	// ************* HMI - Show machine status on main screen ************* //
	IF ("dbUnit".Unit[1].Regime=0) AND NOT "dbUnit".Unit[1].StartStop THEN 
	  "dbUnit".Unit[1].Status     := 1;
	ELSIF ("dbUnit".Unit[1].Regime=0) AND "dbUnit".Unit[1].StartStop THEN 
	  "dbUnit".Unit[1].Status     := 2;
	ELSIF ("dbUnit".Unit[1].Regime>=1) AND NOT "dbUnit".Unit[1].StartStop THEN 
	  "dbUnit".Unit[1].Status     := 3;
	ELSIF ("dbUnit".Unit[1].Regime>=1) AND "dbUnit".Unit[1].StartStop THEN 
	  "dbUnit".Unit[1].Status     := 4;
	ELSIF ("dbUnit".Unit[1].Regime=0) AND ((NOT "ph_Helix_1_DB".InitPosition AND ("ph_Helix_1_DB".CurrentStep > 1 AND "ph_Helix_1_DB".CurrentStep <=2)) OR
	(NOT "ph_LegsShifter_2_DB".InitPosition AND ("ph_LegsShifter_2_DB".CurrentStep > 2 AND "ph_LegsShifter_2_DB".CurrentStep <=3))) THEN
	  "dbUnit".Unit[1].Status     := 5;
	END_IF;
	(*
	1-IZBRAN AVTOMATSKI NAČIN DELOVANJA
	2-AVTOMATSKI NAČIN AKTIVIRAN
	3-IZBRAN ROČNI NAČIN DELOVANJA
	4-ROČNI NAČIN AKTIVIRAN
	5-NAPRAVA NI V IZHODIŠČU
	*)
	// ************* HMI - Show machine status on main screen ************* //
	
	// ************* HMI - Animate HMI button ************* //
	IF "op_ButtonHelix_3_DB".AlarmPresent OR "ph_Helix_1_DB".AlarmPresent OR "ph_LegsShifter_2_DB".AlarmPresent THEN
	  "dbUnit".Unit[1].AlarmsPresent := True;
	ELSE
	  "dbUnit".Unit[1].AlarmsPresent := False;
	END_IF;
	// ************* HMI - Animate HMI button  ************* //
	
	// ************* HMI - BEGIN - Select screen  ************* //
	IF "dbUnit".Unit[1].Regime = 1 AND "dbUnit".Unit[1].StartStop THEN
	  (* NOT IN FUNCTION
	  IF "dbHMIUser".HMICurrScreen = 1 THEN
	    "dbHMIUser".SetTargetHMIScreen    := 2;
	  END_IF;
	  *)
	  IF ("dbHMIUser".HMICurrScreen <> 1) THEN 
	    ; // "dbHMIUser".SetTargetHMIScreen  := 0;
	  END_IF;
	END_IF;
	IF (NOT "dbUnit".Unit[1].StartStop) THEN
	  "dbHMIUser".SetTargetHMIScreen  := 0;
	END_IF;
	"dbHMIUser".HMICurrScreen_OLD := "dbHMIUser".HMICurrScreen;
	// ************* HMI - END - Select screen  ************* //
	
	// ************* HMI - BEGIN - Fill system param  ************* //
	"dbDigitalSensors".KONCNA_POZICIJA_VIJACENJA_DES_NAZAJ.FilterTime       := "dbSystemParam".KONCNA_POZICIJA_VIJACENJA_DES_NAZAJ_FilterTime;
	"dbDigitalSensors".KONCNA_POZICIJA_VIJACENJA_DES_NAPREJ.FilterTime      := "dbSystemParam".KONCNA_POZICIJA_VIJACENJA_DES_NAPREJ_FilterTime;
	"dbDigitalSensors".KONCNA_POZICIJA_VIJACENJA_LEVO_NAZAJ.FilterTime      := "dbSystemParam".KONCNA_POZICIJA_VIJACENJA_LEVO_NAZAJ_FilterTime;
	"dbDigitalSensors".KONCNA_POZICIJA_VIJACENJA_LEVO_NAPREJ.FilterTime     := "dbSystemParam".KONCNA_POZICIJA_VIJACENJA_DES_NAPREJ_FilterTime;
	"op_ButtonHelix_3_DB".DlyTimeToStart_TRAK_VIJAC := "dbSystemParam".DlyTimeToStart_TRAK_VIJAC*10;
	"op_ButtonHelix_3_DB".DlyTimeToStop_TRAK_VIJAC  := "dbSystemParam".DlyTimeToStop_TRAK_VIJAC*10;
	"op_ButtonHelix_3_DB".DlyTimeToStart_VIBRO      := "dbSystemParam".DlyTimeToStart_VIBRO*10;
	"op_ButtonHelix_3_DB".DlyTimeToStop_VIBRO       := "dbSystemParam".DlyTimeToStop_VIBRO*10;
	"dbTimers".Num[8].PRE                           := "dbSystemParam".StandbyTimeTrakaVijac*10*60; // On HMI in unit [min],
	"op_ButtonHelix_3_DB".DlyTimeForAlarmAddNewHelix := "dbSystemParam".DlyTimeForAlarmAddNewHelix * 10;
	// ************* HMI - END - Fill system param  ************* //
	
	// ************* BEGIN - Stop running trak vijačnika, if helix is no more in execution  ************* //
	// See above line "dbTimers".Num[8].PRE                           := "dbSystemParam".StandbyTimeTrakaVijac*10*60; // On HMI in unit [min]
	"dbTimers".Num[8].EE := "dbMotors".VKLOP_M_TRAKA_VIJACNIKA.XS;
	"dbTimers".Num[8].RS := "ph_Helix_1_DB".MovingUPDOWN_Activated;
	
	IF "dbTimers".Num[8].EE AND "dbTimers".Num[8].DN THEN
	  "dbTimers".Num[8].EE := False;
	  "dbTimers".Num[8].DN := False;
	  "dbTimers".Num[8].RS := False;
	  
	  "dbUnit".Unit[1].StartStop := False;
	END_IF;
	// ************* END - Stop running trak vijačnika, if helix is no more in execution  ************* //
END_FUNCTION

FUNCTION "fcDigitalValves" : Void
{ S7_Optimized_Access := 'FALSE' }
VERSION : 0.1
   VAR_TEMP 
      DigitalValveTime : Byte;
   END_VAR


BEGIN
	// Short summary:
	(*
	  Digital valves filter time set, output write and function call
	*)
	// 
	//**********************************************************************
	// Revision control:
	//----------------------------------------------------------------------
	// Use only for revisions of original code
	// V0.01
	// Description of revision
	
	//----------------------------------------------------------------------
	// Comments:
	(*
	  Every change in the code is documented with following:
	  // CCC-yyymmdd: .....
	  yyyy year when change was made
	  mm   month when change was made
	  dd   day when change was made
	  CCC  authors initials
	*)
	
	(*
	- VPENJANJE: V18
	- CENTRIRANJE: V7, V10, V14, V17
	- STOP VIJACENJA ZADAJ: V5, V12
	- LOCEVANJE VIJACENJA: V4, V11
	- LOCEVANJE DRCA: V2, V3
	- DVIG/SPUST VIJACENJA: V6, V9, V13, V16
	*)
	
	//**********************************************************************
	#DigitalValveTime := 10; // Filter time =0. For digital valve is used throught digital sensor with filter time for ."InputF"
	//----------------------------------------------------------------------
	//  set initial values
	"dbDigitalValves".Y17_RotCilipozDesno.FilterTime    := 15;
	"dbDigitalValves".Y18_RotCilipozLevo.FilterTime     := 15;
	"dbDigitalValves".Y2_VijaDesZad_Dvig.FilterTime     := 50;
	"dbDigitalValves".Y3_VijaDesSpr_Dvig.FilterTime     := 50;
	"dbDigitalValves".Y4_VijaLevZad_Dvig.FilterTime     := 50;
	"dbDigitalValves".Y5_VijaLevSpr_Dvig.FilterTime     := 50;
	"dbDigitalValves".Y6_DrcaLocev_Des.FilterTime       := #DigitalValveTime;
	"dbDigitalValves".Y7_DrcaLocev_Lev.FilterTime       := #DigitalValveTime;
	"dbDigitalValves".Y8_VijaLocev_Des.FilterTime       := #DigitalValveTime;
	"dbDigitalValves".Y9_VijaStop_DesZad.FilterTime     := #DigitalValveTime;
	"dbDigitalValves".Y10_Centri_DesZad.FilterTime      := #DigitalValveTime;
	"dbDigitalValves".Y11_Centri_DesSpr.FilterTime      := #DigitalValveTime;
	"dbDigitalValves".Y12_VijaLocev_Lev.FilterTime      := #DigitalValveTime;
	"dbDigitalValves".Y13_VijaStop_LevZad.FilterTime    := #DigitalValveTime;
	"dbDigitalValves".Y14_Centri_LevZad.FilterTime      := #DigitalValveTime;
	"dbDigitalValves".Y15_Centri_LevSpr.FilterTime      := #DigitalValveTime;
	"dbDigitalValves".Y16_VpenjanjeDna.FilterTime       := 30;
	"dbDigitalValves".SEMAFOR_ZELENA.FilterTime         := #DigitalValveTime;
	"dbDigitalValves".SEMAFOR_RUMENA.FilterTime         := #DigitalValveTime;
	"dbDigitalValves".SEMAFOR_RDECA.FilterTime          := #DigitalValveTime;
	
	"dbDigitalValves".Y17_RotCilipozDesno.Invert       := False;
	"dbDigitalValves".Y18_RotCilipozLevo.Invert        := False;
	"dbDigitalValves".Y2_VijaDesZad_Dvig.Invert       := False;
	"dbDigitalValves".Y3_VijaDesSpr_Dvig.Invert       := False;
	"dbDigitalValves".Y4_VijaLevZad_Dvig.Invert      := False;
	"dbDigitalValves".Y5_VijaLevSpr_Dvig.Invert      := False;
	"dbDigitalValves".Y6_DrcaLocev_Des.Invert         := False;
	"dbDigitalValves".Y7_DrcaLocev_Lev.Invert         := False;
	"dbDigitalValves".Y8_VijaLocev_Des.Invert         := False;
	"dbDigitalValves".Y9_VijaStop_DesZad.Invert       := False;
	"dbDigitalValves".Y10_Centri_DesZad.Invert         := False;
	"dbDigitalValves".Y11_Centri_DesSpr.Invert        := False;
	"dbDigitalValves".Y12_VijaLocev_Lev.Invert        := False;
	"dbDigitalValves".Y13_VijaStop_LevZad.Invert      := False;
	"dbDigitalValves".Y14_Centri_LevZad.Invert        := False;
	"dbDigitalValves".Y15_Centri_LevSpr.Invert        := False;
	"dbDigitalValves".Y16_VpenjanjeDna.Invert         := False;
	"dbDigitalValves".SEMAFOR_ZELENA.Invert           := False;
	"dbDigitalValves".SEMAFOR_RUMENA.Invert           := False;
	"dbDigitalValves".SEMAFOR_RDECA.Invert            := False;
	
	"dbDigitalValves".Y17_RotCilipozDesno.AlarmAck       := "AlarmAck";
	"dbDigitalValves".Y18_RotCilipozLevo.AlarmAck        := "AlarmAck";
	"dbDigitalValves".Y2_VijaDesZad_Dvig.AlarmAck       := "AlarmAck";
	"dbDigitalValves".Y3_VijaDesSpr_Dvig.AlarmAck       := "AlarmAck";
	"dbDigitalValves".Y4_VijaLevZad_Dvig.AlarmAck      := "AlarmAck";
	"dbDigitalValves".Y5_VijaLevSpr_Dvig.AlarmAck      := "AlarmAck";
	"dbDigitalValves".Y6_DrcaLocev_Des.AlarmAck         := "AlarmAck";
	"dbDigitalValves".Y7_DrcaLocev_Lev.AlarmAck         := "AlarmAck";
	"dbDigitalValves".Y8_VijaLocev_Des.AlarmAck         := "AlarmAck";
	"dbDigitalValves".Y9_VijaStop_DesZad.AlarmAck       := "AlarmAck";
	"dbDigitalValves".Y10_Centri_DesZad.AlarmAck         := "AlarmAck";
	"dbDigitalValves".Y11_Centri_DesSpr.AlarmAck        := "AlarmAck";
	"dbDigitalValves".Y12_VijaLocev_Lev.AlarmAck        := "AlarmAck";
	"dbDigitalValves".Y13_VijaStop_LevZad.AlarmAck      := "AlarmAck";
	"dbDigitalValves".Y14_Centri_LevZad.AlarmAck        := "AlarmAck";
	"dbDigitalValves".Y15_Centri_LevSpr.AlarmAck        := "AlarmAck";
	"dbDigitalValves".Y16_VpenjanjeDna.AlarmAck         := "AlarmAck";
	"dbDigitalValves".SEMAFOR_ZELENA.AlarmAck           := "AlarmAck";
	"dbDigitalValves".SEMAFOR_RUMENA.AlarmAck           := "AlarmAck";
	"dbDigitalValves".SEMAFOR_RDECA.AlarmAck            := "AlarmAck";
	
	// read GSL
	"dbDigitalValves".Y17_RotCilipozDesno.GSLEnable    := TRUE;
	"dbDigitalValves".Y17_RotCilipozDesno.GSL          := "dbDigitalSensors".ROTACIJSKI_CIL_SREDINA.InputF OR "dbDigitalValves".Y18_RotCilipozLevo.XS;
	"dbDigitalValves".Y18_RotCilipozLevo.GSLEnable     := TRUE;
	"dbDigitalValves".Y18_RotCilipozLevo.GSL           := "dbDigitalSensors".ROTACIJSKI_CIL_SREDINA.InputF OR "dbDigitalValves".Y17_RotCilipozDesno.XS;
	"dbDigitalValves".Y2_VijaDesZad_Dvig.GSLEnable    := True;
	"dbDigitalValves".Y2_VijaDesZad_Dvig.GSL          := "dbDigitalSensors".MESTO_VIJACENJE_DESNO_ZAD_DVIG_DOL.InputF;
	"dbDigitalValves".Y3_VijaDesSpr_Dvig.GSLEnable    := True;
	"dbDigitalValves".Y3_VijaDesSpr_Dvig.GSL          := "dbDigitalSensors".MESTO_VIJACENJE_DESNO_SPRED_DVIG_DOL.InputF;
	"dbDigitalValves".Y4_VijaLevZad_Dvig.GSLEnable   := True;
	"dbDigitalValves".Y4_VijaLevZad_Dvig.GSL         := "dbDigitalSensors".MESTO_VIJACENJE_LEVO_ZAD_DVIG_DOL.InputF;
	"dbDigitalValves".Y5_VijaLevSpr_Dvig.GSLEnable   := True;
	"dbDigitalValves".Y5_VijaLevSpr_Dvig.GSL         := "dbDigitalSensors".MESTO_VIJACENJE_LEVO_SPRED_DVIG_DOL.InputF;
	"dbDigitalValves".Y6_DrcaLocev_Des.GSLEnable      := True;
	"dbDigitalValves".Y6_DrcaLocev_Des.GSL            := "dbDigitalSensors".LOC_DRCA_DESNO_NAPREJ.InputF;
	"dbDigitalValves".Y7_DrcaLocev_Lev.GSLEnable      := True;
	"dbDigitalValves".Y7_DrcaLocev_Lev.GSL            := "dbDigitalSensors".LOC_DRCA_LEVO_NAPREJ.InputF;
	"dbDigitalValves".Y8_VijaLocev_Des.GSLEnable      := True;
	"dbDigitalValves".Y8_VijaLocev_Des.GSL            := "dbDigitalSensors".VIJACENJE_DESNO_1_NAPREJ.InputF;
	"dbDigitalValves".Y9_VijaStop_DesZad.GSLEnable    := True;
	"dbDigitalValves".Y9_VijaStop_DesZad.GSL          := "dbDigitalSensors".MESTO_VIJAC_STOP_DESNO_ZAD_NAPREJ.InputF;
	"dbDigitalValves".Y10_Centri_DesZad.GSLEnable      := True;
	"dbDigitalValves".Y10_Centri_DesZad.GSL            := "dbDigitalSensors".MESTO_VIJACENJE_DESNO_ZAD_CENT_NARAZEN.InputF;
	"dbDigitalValves".Y11_Centri_DesSpr.GSLEnable     := True;
	"dbDigitalValves".Y11_Centri_DesSpr.GSL           := "dbDigitalSensors".MESTO_VIJACENJE_DESNO_SPRED_CENT_NARAZEN.InputF;
	"dbDigitalValves".Y12_VijaLocev_Lev.GSLEnable     := True;
	"dbDigitalValves".Y12_VijaLocev_Lev.GSL           := "dbDigitalSensors".VIJACENJE_LEVO_1_NAPREJ.InputF;
	"dbDigitalValves".Y13_VijaStop_LevZad.GSLEnable   := True;
	"dbDigitalValves".Y13_VijaStop_LevZad.GSL         := "dbDigitalSensors".MESTO_VIJAC_STOP_LEVO_ZAD_NAPREJ.InputF;
	"dbDigitalValves".Y14_Centri_LevZad.GSLEnable     := True;
	"dbDigitalValves".Y14_Centri_LevZad.GSL           := "dbDigitalSensors".MESTO_VIJACENJE_LEVO_ZAD_CENT_NARAZEN.InputF;
	"dbDigitalValves".Y15_Centri_LevSpr.GSLEnable     := True;
	"dbDigitalValves".Y15_Centri_LevSpr.GSL           := "dbDigitalSensors".MESTO_VIJACENJE_LEVO_SPRED_CENT_NARAZEN.InputF;
	"dbDigitalValves".Y16_VpenjanjeDna.GSLEnable      := True;
	"dbDigitalValves".Y16_VpenjanjeDna.GSL            := "dbDigitalSensors".VPENJANJE_DNA_LEVO_ZADAJ_GOR.InputF AND "dbDigitalSensors".VPENJANJE_DNA_LEVO_SPREDAJ_GOR.InputF AND
	                                                     "dbDigitalSensors".VPENJANJE_DNA_DESNO_ZADAJ_GOR.InputF AND "dbDigitalSensors".VPENJANJE_DNA_DESNO_SPREDAJ_GOR.InputF;
	
	// read GSH
	"dbDigitalValves".Y17_RotCilipozDesno.GSHEnable    := TRUE;
	"dbDigitalValves".Y17_RotCilipozDesno.GSH          := "dbDigitalSensors".ROTACIJSKI_CIL_DESNO.InputF;
	"dbDigitalValves".Y18_RotCilipozLevo.GSHEnable     := True;
	"dbDigitalValves".Y18_RotCilipozLevo.GSH           := "dbDigitalSensors".ROTACIJSKI_CIL_LEVO.InputF;
	"dbDigitalValves".Y2_VijaDesZad_Dvig.GSHEnable    := FALSE;
	"dbDigitalValves".Y2_VijaDesZad_Dvig.GSH          := FALSE;
	"dbDigitalValves".Y3_VijaDesSpr_Dvig.GSHEnable    := FALSE;
	"dbDigitalValves".Y3_VijaDesSpr_Dvig.GSH          := FALSE;
	"dbDigitalValves".Y4_VijaLevZad_Dvig.GSHEnable   := FALSE;
	"dbDigitalValves".Y4_VijaLevZad_Dvig.GSH         := FALSE;
	"dbDigitalValves".Y5_VijaLevSpr_Dvig.GSHEnable   := False;
	"dbDigitalValves".Y5_VijaLevSpr_Dvig.GSH         := False;
	"dbDigitalValves".Y6_DrcaLocev_Des.GSHEnable      := True;
	"dbDigitalValves".Y6_DrcaLocev_Des.GSH            := "dbDigitalSensors".LOC_DRCA_DESNO_NAZAJ.InputF;
	"dbDigitalValves".Y7_DrcaLocev_Lev.GSHEnable      := True;
	"dbDigitalValves".Y7_DrcaLocev_Lev.GSH            := "dbDigitalSensors".LOC_DRCA_LEVO_NAZAJ.InputF;
	"dbDigitalValves".Y8_VijaLocev_Des.GSHEnable      := True;
	"dbDigitalValves".Y8_VijaLocev_Des.GSH            := "dbDigitalSensors".VIJACENJE_DESNO_1_NAZAJ.InputF;
	"dbDigitalValves".Y9_VijaStop_DesZad.GSHEnable    := True;
	"dbDigitalValves".Y9_VijaStop_DesZad.GSH          := "dbDigitalSensors".MESTO_VIJAC_STOP_DESNO_ZAD_NAZAJ.InputF;
	"dbDigitalValves".Y10_Centri_DesZad.GSHEnable      := True;
	"dbDigitalValves".Y10_Centri_DesZad.GSH            := "dbDigitalSensors".MESTO_VIJACENJE_DESNO_ZAD_CENT_SKUPAJ.InputF;
	"dbDigitalValves".Y11_Centri_DesSpr.GSHEnable     := True;
	"dbDigitalValves".Y11_Centri_DesSpr.GSH           := "dbDigitalSensors".MESTO_VIJACENJE_DESNO_SPRED_CENT_SKUPAJ.InputF;
	"dbDigitalValves".Y12_VijaLocev_Lev.GSHEnable     := True;
	"dbDigitalValves".Y12_VijaLocev_Lev.GSH           := "dbDigitalSensors".VIJACENJE_LEVO_1_NAZAJ.InputF;
	"dbDigitalValves".Y13_VijaStop_LevZad.GSHEnable   := True;
	"dbDigitalValves".Y13_VijaStop_LevZad.GSH         := "dbDigitalSensors".MESTO_VIJAC_STOP_LEVO_ZAD_NAZAJ.InputF;;
	"dbDigitalValves".Y14_Centri_LevZad.GSHEnable     := True;
	"dbDigitalValves".Y14_Centri_LevZad.GSH           := "dbDigitalSensors".MESTO_VIJACENJE_LEVO_ZAD_CENT_SKUPAJ.InputF;
	"dbDigitalValves".Y15_Centri_LevSpr.GSHEnable     := True;
	"dbDigitalValves".Y15_Centri_LevSpr.GSH           := "dbDigitalSensors".MESTO_VIJACENJE_LEVO_SPRED_CENT_SKUPAJ.InputF;
	"dbDigitalValves".Y16_VpenjanjeDna.GSHEnable      := True;
	"dbDigitalValves".Y16_VpenjanjeDna.GSH            := "dbDigitalSensors".VPENJANJE_DNA_LEVO_ZADAJ_DOL.InputF AND "dbDigitalSensors".VPENJANJE_DNA_LEVO_SPREDAJ_DOL.InputF AND
	                                                     "dbDigitalSensors".VPENJANJE_DNA_DESNO_ZADAJ_DOL.InputF AND "dbDigitalSensors".VPENJANJE_DNA_DESNO_SPREDAJ_DOL.InputF;
	
	// Reset Manual Regime, if selected AUTO regime on HMI
	//----------------------------------------------------------------------
	IF "dbUnit".Unit[1].Regime = 0 AND "dbUnit".Unit[1].StartStop THEN
	  "dbDigitalValves".Y17_RotCilipozDesno.ManON   := False;
	  "dbDigitalValves".Y18_RotCilipozLevo.ManON    := False;
	  "dbDigitalValves".Y2_VijaDesZad_Dvig.ManON    := False;
	  "dbDigitalValves".Y2_VijaDesZad_Dvig.ManON    := False;
	  "dbDigitalValves".Y3_VijaDesSpr_Dvig.ManON    := False;
	  "dbDigitalValves".Y3_VijaDesSpr_Dvig.ManON    := False;
	  "dbDigitalValves".Y4_VijaLevZad_Dvig.ManON    := False;
	  "dbDigitalValves".Y4_VijaLevZad_Dvig.ManON    := False;
	  "dbDigitalValves".Y5_VijaLevSpr_Dvig.ManON    := False;
	  "dbDigitalValves".Y5_VijaLevSpr_Dvig.ManON    := False;
	  "dbDigitalValves".Y6_DrcaLocev_Des.ManON      := False;
	  "dbDigitalValves".Y7_DrcaLocev_Lev.ManON      := False;
	  "dbDigitalValves".Y8_VijaLocev_Des.ManON      := False;
	  "dbDigitalValves".Y9_VijaStop_DesZad.ManON    := False;
	  "dbDigitalValves".Y10_Centri_DesZad.ManON     := False;
	  "dbDigitalValves".Y11_Centri_DesSpr.ManON     := False;
	  "dbDigitalValves".Y12_VijaLocev_Lev.ManON     := False;
	  "dbDigitalValves".Y13_VijaStop_LevZad.ManON   := False;
	  "dbDigitalValves".Y14_Centri_LevZad.ManON     := False;
	  "dbDigitalValves".Y15_Centri_LevSpr.ManON     := False;
	ELSIF "dbUnit".Unit[1].Regime = 1 AND NOT "dbUnit".Unit[1].StartStop THEN
	  "dbDigitalValves".Y17_RotCilipozDesno.ManON   := False;
	  "dbDigitalValves".Y18_RotCilipozLevo.ManON    := False;
	  "dbDigitalValves".Y2_VijaDesZad_Dvig.ManON    := False;
	  "dbDigitalValves".Y2_VijaDesZad_Dvig.ManON    := False;
	  "dbDigitalValves".Y3_VijaDesSpr_Dvig.ManON    := False;
	  "dbDigitalValves".Y3_VijaDesSpr_Dvig.ManON    := False;
	  "dbDigitalValves".Y4_VijaLevZad_Dvig.ManON    := False;
	  "dbDigitalValves".Y4_VijaLevZad_Dvig.ManON    := False;
	  "dbDigitalValves".Y5_VijaLevSpr_Dvig.ManON    := False;
	  "dbDigitalValves".Y5_VijaLevSpr_Dvig.ManON    := False;
	  "dbDigitalValves".Y6_DrcaLocev_Des.ManON      := False;
	  "dbDigitalValves".Y7_DrcaLocev_Lev.ManON      := False;
	  "dbDigitalValves".Y8_VijaLocev_Des.ManON      := False;
	  "dbDigitalValves".Y9_VijaStop_DesZad.ManON    := False;
	  "dbDigitalValves".Y10_Centri_DesZad.ManON     := False;
	  "dbDigitalValves".Y11_Centri_DesSpr.ManON     := False;
	  "dbDigitalValves".Y12_VijaLocev_Lev.ManON     := False;
	  "dbDigitalValves".Y13_VijaStop_LevZad.ManON   := False;
	  "dbDigitalValves".Y14_Centri_LevZad.ManON     := False;
	  "dbDigitalValves".Y15_Centri_LevSpr.ManON     := False;
	END_IF; 
	
	//----------------------------------------------------------------------
	// fc call
	"cmDigitalValve"(Regime := "dbUnit".Unit[1].Regime, Valve := "dbDigitalValves".Y17_RotCilipozDesno);
	"cmDigitalValve"(Regime := "dbUnit".Unit[1].Regime, Valve := "dbDigitalValves".Y18_RotCilipozLevo);
	"cmDigitalValve"(Regime := "dbUnit".Unit[1].Regime, Valve := "dbDigitalValves".Y2_VijaDesZad_Dvig);
	"cmDigitalValve"(Regime := "dbUnit".Unit[1].Regime, Valve := "dbDigitalValves".Y3_VijaDesSpr_Dvig);
	"cmDigitalValve"(Regime := "dbUnit".Unit[1].Regime, Valve := "dbDigitalValves".Y4_VijaLevZad_Dvig);
	"cmDigitalValve"(Regime := "dbUnit".Unit[1].Regime, Valve := "dbDigitalValves".Y5_VijaLevSpr_Dvig);
	"cmDigitalValve"(Regime := "dbUnit".Unit[1].Regime, Valve := "dbDigitalValves".Y6_DrcaLocev_Des);
	"cmDigitalValve"(Regime := "dbUnit".Unit[1].Regime, Valve := "dbDigitalValves".Y7_DrcaLocev_Lev);
	"cmDigitalValve"(Regime := "dbUnit".Unit[1].Regime, Valve := "dbDigitalValves".Y8_VijaLocev_Des);
	"cmDigitalValve"(Regime := "dbUnit".Unit[1].Regime, Valve := "dbDigitalValves".Y9_VijaStop_DesZad);
	"cmDigitalValve"(Regime := "dbUnit".Unit[1].Regime, Valve := "dbDigitalValves".Y10_Centri_DesZad);
	"cmDigitalValve"(Regime := "dbUnit".Unit[1].Regime, Valve := "dbDigitalValves".Y11_Centri_DesSpr);
	"cmDigitalValve"(Regime := "dbUnit".Unit[1].Regime, Valve := "dbDigitalValves".Y12_VijaLocev_Lev);
	"cmDigitalValve"(Regime := "dbUnit".Unit[1].Regime, Valve := "dbDigitalValves".Y13_VijaStop_LevZad);
	"cmDigitalValve"(Regime := "dbUnit".Unit[1].Regime, Valve := "dbDigitalValves".Y14_Centri_LevZad);
	"cmDigitalValve"(Regime := "dbUnit".Unit[1].Regime, Valve := "dbDigitalValves".Y15_Centri_LevSpr);
	"cmDigitalValve"(Regime := "dbUnit".Unit[1].Regime, Valve := "dbDigitalValves".Y16_VpenjanjeDna);
	"cmDigitalValve"(Regime := "dbUnit".Unit[1].Regime, Valve := "dbDigitalValves".SEMAFOR_ZELENA);
	"cmDigitalValve"(Regime := "dbUnit".Unit[1].Regime, Valve := "dbDigitalValves".SEMAFOR_RUMENA);
	"cmDigitalValve"(Regime := "dbUnit".Unit[1].Regime, Valve := "dbDigitalValves".SEMAFOR_RDECA);
	
	//----------------------------------------------------------------------
	//  write output
	"dbPDO".Y17_RotCilipozDesno    := "dbDigitalValves".Y17_RotCilipozDesno.XS;
	"dbPDO".Y18_RotCilipozLevo     := "dbDigitalValves".Y18_RotCilipozLevo.XS;
	"dbPDO".Y2_VijaDesZad_Dvig    := "dbDigitalValves".Y2_VijaDesZad_Dvig.XS;
	"dbPDO".Y2_VijaDesZad_Spust   := NOT "dbDigitalValves".Y2_VijaDesZad_Dvig.XS;
	"dbPDO".Y3_VijaDesSpr_Dvig    := "dbDigitalValves".Y3_VijaDesSpr_Dvig.XS;
	"dbPDO".Y3_VijaDesSpr_Spust   := NOT "dbDigitalValves".Y3_VijaDesSpr_Dvig.XS;
	"dbPDO".Y4_VijaLevZad_Dvig   := "dbDigitalValves".Y4_VijaLevZad_Dvig.XS;
	"dbPDO".Y4_VijaLevZad_Spust  := NOT "dbDigitalValves".Y4_VijaLevZad_Dvig.XS;
	"dbPDO".Y5_VijaLevSpr_Dvig   := "dbDigitalValves".Y5_VijaLevSpr_Dvig.XS;
	"dbPDO".Y5_VijaLevSpr_Spust  := NOT "dbDigitalValves".Y5_VijaLevSpr_Dvig.XS;
	"dbPDO".Y6_DrcaLocev_Des      := "dbDigitalValves".Y6_DrcaLocev_Des.XS;
	"dbPDO".Y7_DrcaLocev_Lev      := "dbDigitalValves".Y7_DrcaLocev_Lev.XS;
	"dbPDO".Y8_VijaLocev_Des      := "dbDigitalValves".Y8_VijaLocev_Des.XS;
	"dbPDO".Y9_VijaStop_DesZad    := "dbDigitalValves".Y9_VijaStop_DesZad.XS;
	"dbPDO".Y10_Centri_DesZad      := "dbDigitalValves".Y10_Centri_DesZad.XS;
	"dbPDO".Y11_Centri_DesSpr     := "dbDigitalValves".Y11_Centri_DesSpr.XS;
	"dbPDO".Y12_VijaLocev_Lev     := "dbDigitalValves".Y12_VijaLocev_Lev.XS;
	"dbPDO".Y13_VijaStop_LevZad   := "dbDigitalValves".Y13_VijaStop_LevZad.XS;
	"dbPDO".Y14_Centri_LevZad     := "dbDigitalValves".Y14_Centri_LevZad.XS;
	"dbPDO".Y15_Centri_LevSpr     := "dbDigitalValves".Y15_Centri_LevSpr.XS;
	"dbPDO".Y16_VpenjanjeDna      := "dbDigitalValves".Y16_VpenjanjeDna.XS;
	
	"dbDO".SEMAFOR_ZELENA         := "dbDigitalValves".SEMAFOR_ZELENA.XS;
	"dbDO".SEMAFOR_RUMENA         := "dbDigitalValves".SEMAFOR_RUMENA.XS;
	"dbDO".SEMAFOR_RDECA          := "dbDigitalValves".SEMAFOR_RDECA.XS;
END_FUNCTION

FUNCTION "cmDigitalValve" : Void
{ S7_Optimized_Access := 'FALSE' }
VERSION : 0.1
   VAR_IN_OUT 
      Regime : USInt;
      Valve : "udtDigitalValve";
   END_VAR

   VAR_TEMP 
      tmpTimer : Int;
      tmpTimerDelay : Int;
   END_VAR

   VAR CONSTANT 
      AlarmAutoResetDly : UInt := 50;
   END_VAR


BEGIN
	// ALARMING
	#tmpTimer := CHAR_TO_INT(BYTE_TO_CHAR(#Valve.Timer1));
	#tmpTimerDelay := CHAR_TO_INT(BYTE_TO_CHAR(#Valve.FilterTime));
	
	IF (NOT #Valve.GSLEnable AND NOT #Valve.GSHEnable) THEN
	    #Valve.Alarm := FALSE;
	    #tmpTimer := 0;
	END_IF;
	
	IF ((#Valve.GSLEnable AND NOT #Valve.GSHEnable) AND ((NOT #Valve.SCADAVis AND NOT #Valve.GSL) OR (#Valve.SCADAVis AND #Valve.GSL))) OR
	    ((NOT #Valve.GSLEnable AND #Valve.GSHEnable) AND ((#Valve.SCADAVis AND NOT #Valve.GSH) OR (NOT #Valve.SCADAVis AND #Valve.GSH))) OR
	    ((#Valve.GSLEnable AND #Valve.GSHEnable) AND ((#Valve.SCADAVis AND (#Valve.GSL OR NOT #Valve.GSH)) OR (NOT #Valve.SCADAVis AND (NOT #Valve.GSL OR #Valve.GSH)))) THEN
	    
	    IF (NOT #Valve.Alarm) AND "100msOSR" AND (#tmpTimer <= #tmpTimerDelay) THEN
	        #tmpTimer := #tmpTimer + 1;
	        IF #tmpTimer >= #tmpTimerDelay THEN
	            #Valve.Alarm := TRUE;
	            #Valve.GSLAlarm := ((#Valve.GSLEnable) AND ((NOT #Valve.SCADAVis AND NOT #Valve.GSL) OR (#Valve.SCADAVis AND #Valve.GSL)));
	            #Valve.GSHAlarm := ((#Valve.GSHEnable) AND ((#Valve.SCADAVis AND NOT #Valve.GSH) OR (NOT #Valve.SCADAVis AND #Valve.GSH)));
	            #tmpTimer := 0;
	        END_IF;
	    END_IF;
	    IF (#Valve.Alarm) THEN
	        #tmpTimer := 0;
	    END_IF;
	// ELSIF ((#Valve.GSLEnable AND NOT #Valve.GSHEnable) AND (NOT #Valve.SCADAVis AND #Valve.GSL) OR // 20210429_PRA
	   ELSIF ((#Valve.GSLEnable AND NOT #Valve.GSHEnable) AND (NOT #Valve.SCADAVis AND #Valve.GSL) OR #Valve.SCADAVis) OR // 20210429_PRA-added to reset timer when valve activated
	    ((NOT #Valve.GSLEnable AND #Valve.GSHEnable) AND (#Valve.SCADAVis AND #Valve.GSH)) OR
	    ((#Valve.GSLEnable AND #Valve.GSHEnable) AND ((#Valve.SCADAVis AND #Valve.GSH) OR (NOT #Valve.SCADAVis AND #Valve.GSL))) THEN
	   
	    #tmpTimer := 0;
	    ;
	    (*
	    IF (#Valve.Alarm) AND "100msOSR" AND (#tmpTimer < AlarmAutoResetDly) THEN // Auto-reset of the alarm after 5 seconds
	        #tmpTimer := #tmpTimer + 1;
	        IF #tmpTimer >= AlarmAutoResetDly THEN
	            #Valve.Alarm := FALSE;
	            #Valve.GSLAlarm := FALSE;
	            #Valve.GSHAlarm := FALSE;
	            #tmpTimer := 0;
	        END_IF;
	    END_IF;
	    IF (NOT #Valve.Alarm) THEN
	        #tmpTimer := 0;
	    END_IF;
	    *)
	END_IF;
	
	//  ALARMING MODULE
	IF #Valve.AlarmAck THEN
	    #Valve.Alarm := FALSE;
	    #Valve.GSLAlarm := FALSE;
	    #Valve.GSHAlarm := FALSE;
	    #Valve.AlarmAck := FALSE;
	    
	    #tmpTimer := 0;
	END_IF;
	
	#Valve.Timer1 := CHAR_TO_BYTE(INT_TO_CHAR(#tmpTimer));
	
	//----------------------------------------------------------------------
	//  OUTPUT   
	#Valve.XS := FALSE;
	
	IF #Regime = 0 THEN
	    #Valve.ManON := FALSE;
	    #Valve.ManOFF := FALSE;
	    #Valve.XS := #Valve.AutoON;
	    #Valve.HMICmd := false;
	ELSIF #Regime > 0 THEN
	    IF #Valve.HMICmd THEN
	        IF NOT #Valve.SCADAVis THEN
	            #Valve.ManON := true;
	            #Valve.ManOFF := false;
	        END_IF;
	        IF #Valve.SCADAVis THEN
	            #Valve.ManON := false;
	            #Valve.ManOFF := true;
	        END_IF;
	        #Valve.HMICmd := false;
	    END_IF;
	    #Valve.XS := (#Valve.AutoON AND NOT #Valve.ManON AND NOT #Valve.ManOFF) OR (#Valve.ManON AND NOT #Valve.ManOFF);
	END_IF;
	
	//----------------------------------------------------------------------
	//  MANUAL BIT
	#Valve.Manual := #Valve.ManON OR #Valve.ManOFF;
	
	//----------------------------------------------------------------------
	//  INTERLOCK
	IF (#Valve.Interlock AND #Regime < 2) THEN
	    #Valve.XS := FALSE;
	END_IF;
	
	//----------------------------------------------------------------------
	//  NORMALY OPEN VALVES
	IF (#Valve.Invert) THEN
	    #Valve.XS := NOT (#Valve.XS);
	END_IF;
	
	//----------------------------------------------------------------------
	// SCADA VIS flag
	IF #Valve.Invert = TRUE THEN
	    #Valve.SCADAVis := NOT (#Valve.XS);
	ELSE
	    #Valve.SCADAVis := #Valve.XS;
	END_IF;
	
	//----------------------------------------------------------------------
	// Valve Status
	IF NOT #Valve.SCADAVis THEN
	    #Valve.Status := 0;
	END_IF;
	IF #Valve.SCADAVis THEN
	    #Valve.Status := 1;
	END_IF;
	IF #Valve.Alarm THEN
	    #Valve.Status := 2;
	END_IF;
	(*
	IF #Valve.GSLAlarm THEN
	    #Valve.Status := 3;
	END_IF;
	IF #Valve.GSHAlarm THEN
	    #Valve.Status := 4;
	END_IF;
	*)
	
	
END_FUNCTION

FUNCTION "fcMotors" : Void
{ S7_Optimized_Access := 'TRUE' }
VERSION : 0.1
   VAR CONSTANT 
      CONST_FILTER_TIME_EA : USInt := 10;
      CONST_FILTER_TIME_FSL : USInt := 50;
   END_VAR


BEGIN
	// Short summary:
	(*
	  fcMotors - call motors
	*)
	// 
	//**********************************************************************
	// Revision control:
	//----------------------------------------------------------------------
	// Use only for revisions of original code
	// V0.01
	// Description of revision
	
	//----------------------------------------------------------------------
	// Comments:
	(*
	  Every change in the code is documented with following:
	  // CCC-yyymmdd: .....
	  yyyy year when change was made
	  mm   month when change was made
	  dd   day when change was made
	  CCC  authors initials
	*)
	//**********************************************************************
	
	//  set motor parameters
	"dbMotors".VKLOP_M_TRACNEGA_TRANS_NOGIC.MaxEng  := 100.0; // Max motor RPM
	"dbMotors".VKLOP_M_TRACNEGA_TRANS_NOGIC.MinEng  := 0.0;   // Min motor RPM
	"dbMotors".VKLOP_M_TRACNEGA_TRANS_NOGIC.ESA     := NOT "dbDigitalSensors".BIMETAL_TRANSPORTA_NOGIC_IZKLJUCIL.InputF;
	"dbMotors".VKLOP_M_TRACNEGA_TRANS_NOGIC.EA      := "dbDO".VKLOP_M_TRACNEGA_TRANS_NOGIC;
	"dbMotors".VKLOP_M_TRACNEGA_TRANS_NOGIC.FSL     := "dbDO".VKLOP_M_TRACNEGA_TRANS_NOGIC;
	"dbMotors".VKLOP_M_TRACNEGA_TRANS_NOGIC.AlarmAck := "AlarmAck";
	// "dbDO". := "dbMotors".M_TRACNEGA_TRANSPORTA.ResetFCAlarm;
	"dbMotors".VKLOP_M_TRACNEGA_TRANS_NOGIC.FILTER_TIME_EA  := #CONST_FILTER_TIME_EA;   // 10 sec
	"dbMotors".VKLOP_M_TRACNEGA_TRANS_NOGIC.FILTER_TIME_FSL := #CONST_FILTER_TIME_FSL;  // 50 sec
	
	"dbMotors".M1_ZADAJ_DESNO.MaxEng  := 100.0; // Max motor RPM
	"dbMotors".M1_ZADAJ_DESNO.MinEng  := 0.0;   // Min motor RPM
	"dbMotors".M1_ZADAJ_DESNO.ESA     := "dbDigitalSensors".FR_MOTORJA1_ZADAJ_DESNO_READY.InputF;
	"dbMotors".M1_ZADAJ_DESNO.EA      := "dbMotors".M1_ZADAJ_DESNO.XS;
	"dbMotors".M1_ZADAJ_DESNO.FSL     := "dbMotors".M1_ZADAJ_DESNO.XS;
	"dbMotors".M1_ZADAJ_DESNO.AlarmAck:= "AlarmAck";
	"dbDO".MOTOR_1_ZADAJ_DESNO_RESET  := "dbMotors".M1_ZADAJ_DESNO.ResetFCAlarm;
	"dbMotors".M1_ZADAJ_DESNO.FILTER_TIME_EA    := #CONST_FILTER_TIME_EA;   // 10 sec
	"dbMotors".M1_ZADAJ_DESNO.FILTER_TIME_FSL   := #CONST_FILTER_TIME_FSL;  // 50 sec
	// Check "dbMotors".M1_ZADAJ_DESNO.Alarm       := False;
	
	"dbMotors".M2_SPREDAJ_DESNO.MaxEng := 100.0; // Max motor RPM
	"dbMotors".M2_SPREDAJ_DESNO.MinEng := 0.0;   // Min motor RPM
	"dbMotors".M2_SPREDAJ_DESNO.ESA := "dbDigitalSensors".FR_MOTORJA2_SPREDAJ_DESNO_READY.InputF;
	"dbMotors".M2_SPREDAJ_DESNO.EA := "dbMotors".M2_SPREDAJ_DESNO.XS;
	"dbMotors".M2_SPREDAJ_DESNO.FSL := "dbMotors".M2_SPREDAJ_DESNO.XS;
	"dbMotors".M2_SPREDAJ_DESNO.AlarmAck := "AlarmAck";
	"dbDO".MOTOR_2_SPREDAJ_DESNO_RESET := "dbMotors".M2_SPREDAJ_DESNO.ResetFCAlarm;
	"dbMotors".M2_SPREDAJ_DESNO.FILTER_TIME_EA := #CONST_FILTER_TIME_EA;   // 10 sec
	"dbMotors".M2_SPREDAJ_DESNO.FILTER_TIME_FSL := #CONST_FILTER_TIME_FSL;  // 50 sec
	// Check "dbMotors".M2_SPREDAJ_DESNO.Alarm       := False; // Check
	
	"dbMotors".M1_ZADAJ_LEVO.MaxEng := 100.0; // Max motor RPM
	"dbMotors".M1_ZADAJ_LEVO.MinEng := 0.0;   // Min motor RPM
	"dbMotors".M1_ZADAJ_LEVO.ESA := "dbDigitalSensors".FR_MOTORJA1_ZADAJ_LEVO_READY.InputF;
	"dbMotors".M1_ZADAJ_LEVO.EA := "dbMotors".M1_ZADAJ_LEVO.XS;
	"dbMotors".M1_ZADAJ_LEVO.FSL := "dbMotors".M1_ZADAJ_LEVO.XS;
	"dbMotors".M1_ZADAJ_LEVO.AlarmAck := "AlarmAck";
	"dbDO".MOTOR_1_ZADAJ_LEVO_RESET := "dbMotors".M1_ZADAJ_LEVO.ResetFCAlarm;
	"dbMotors".M1_ZADAJ_LEVO.FILTER_TIME_EA := #CONST_FILTER_TIME_EA;   // 10 sec
	"dbMotors".M1_ZADAJ_LEVO.FILTER_TIME_FSL := #CONST_FILTER_TIME_FSL;  // 50 sec
	// Check "dbMotors".M1_ZADAJ_LEVO.Alarm       := False; // Check
	
	"dbMotors".M2_SPREDAJ_LEVO.MaxEng := 100.0; // Max motor RPM
	"dbMotors".M2_SPREDAJ_LEVO.MinEng := 0.0;   // Min motor RPM
	"dbMotors".M2_SPREDAJ_LEVO.ESA := "dbDigitalSensors".FR_MOTORJA2_SPREDAJ_LEVO_READY.InputF;
	"dbMotors".M2_SPREDAJ_LEVO.EA := "dbMotors".M2_SPREDAJ_LEVO.XS;
	"dbMotors".M2_SPREDAJ_LEVO.FSL := "dbMotors".M2_SPREDAJ_LEVO.XS;
	"dbMotors".M2_SPREDAJ_LEVO.AlarmAck := "AlarmAck";
	"dbDO".MOTOR_2_SPREDAJ_LEVO_RESET := "dbMotors".M2_SPREDAJ_LEVO.ResetFCAlarm;
	"dbMotors".M2_SPREDAJ_LEVO.FILTER_TIME_EA := #CONST_FILTER_TIME_EA;   // 10 sec
	"dbMotors".M2_SPREDAJ_LEVO.FILTER_TIME_FSL := #CONST_FILTER_TIME_FSL;  // 50 sec
	// Check "dbMotors".M2_SPREDAJ_LEVO.Alarm       := False; // Check
	
	"dbMotors".VKLOP_VIBRATORJA.MaxEng := 100.0; // Max motor RPM
	"dbMotors".VKLOP_VIBRATORJA.MinEng := 0.0;   // Min motor RPM
	"dbMotors".VKLOP_VIBRATORJA.ESA := TRUE;
	"dbMotors".VKLOP_VIBRATORJA.EA := "dbDO".VKLOP_VIBRATORJA; // NOT EL. INSTALLED "dbDigitalSensors".VIBRATOR_NOGIC_READY.InputF
	"dbMotors".VKLOP_VIBRATORJA.FSL := "dbDO".VKLOP_VIBRATORJA;
	"dbMotors".VKLOP_VIBRATORJA.AlarmAck := "AlarmAck";
	// "dbDO". := "dbMotors".VKLOP_VIBRATORJA.ResetFCAlarm;
	"dbMotors".VKLOP_VIBRATORJA.FILTER_TIME_EA := #CONST_FILTER_TIME_EA;   // 10 sec
	"dbMotors".VKLOP_VIBRATORJA.FILTER_TIME_FSL := #CONST_FILTER_TIME_FSL;  // 50 sec
	
	"dbMotors".VKLOP_M_TRAKA_VIJACNIKA.MaxEng := 100.0; // Max motor RPM
	"dbMotors".VKLOP_M_TRAKA_VIJACNIKA.MinEng := 0.0;   // Min motor RPM
	"dbMotors".VKLOP_M_TRAKA_VIJACNIKA.ESA :=  NOT "dbDigitalSensors".BIMETAL_VIJACENJA_NOGIC_IZKLJUCIL.InputF;
	"dbMotors".VKLOP_M_TRAKA_VIJACNIKA.EA := "dbDO".VKLOP_M_TRAKA_VIJACNIKA;
	"dbMotors".VKLOP_M_TRAKA_VIJACNIKA.FSL := "dbDO".VKLOP_M_TRAKA_VIJACNIKA;
	"dbMotors".VKLOP_M_TRAKA_VIJACNIKA.AlarmAck := "AlarmAck";
	// "dbDO". := "dbMotors".VKLOP_M_TRAKA_VIJACNIKA.ResetFCAlarm;
	"dbMotors".VKLOP_M_TRAKA_VIJACNIKA.FILTER_TIME_EA := #CONST_FILTER_TIME_EA;   // 10 sec
	"dbMotors".VKLOP_M_TRAKA_VIJACNIKA.FILTER_TIME_FSL := #CONST_FILTER_TIME_FSL;  // 50 sec
	
	// Reset Manual Regime, if selected AUTO regime on HMI
	//----------------------------------------------------------------------
	IF "dbUnit".Unit[1].Regime = 0 AND "dbUnit".Unit[1].StartStop THEN
	  "dbMotors".VKLOP_M_TRACNEGA_TRANS_NOGIC.ManON   := False;
	  "dbMotors".M1_ZADAJ_DESNO.ManON                 := False;
	  "dbMotors".M2_SPREDAJ_DESNO.ManON               := False;
	  "dbMotors".M1_ZADAJ_LEVO.ManON                  := False;
	  "dbMotors".M2_SPREDAJ_LEVO.ManON                := False;
	  "dbMotors".VKLOP_VIBRATORJA.ManON               := False;
	  "dbMotors".VKLOP_M_TRAKA_VIJACNIKA.ManON        := False;
	ELSIF "dbUnit".Unit[1].Regime = 1 AND NOT "dbUnit".Unit[1].StartStop THEN
	  "dbMotors".VKLOP_M_TRACNEGA_TRANS_NOGIC.ManON   := False;
	  "dbMotors".M1_ZADAJ_DESNO.ManON                 := False;
	  "dbMotors".M2_SPREDAJ_DESNO.ManON               := False;
	  "dbMotors".M1_ZADAJ_LEVO.ManON                  := False;
	  "dbMotors".M2_SPREDAJ_LEVO.ManON                := False;
	  "dbMotors".VKLOP_VIBRATORJA.ManON               := False;
	  "dbMotors".VKLOP_M_TRAKA_VIJACNIKA.ManON        := False;
	END_IF;
	
	//----------------------------------------------------------------------
	// fc call
	"cmMotor"(Regime := "dbUnit".Unit[1].Regime, FQ := "dbMotors".VKLOP_M_TRACNEGA_TRANS_NOGIC);
	"cmMotor"(Regime := "dbUnit".Unit[1].Regime, FQ := "dbMotors".M1_ZADAJ_DESNO);
	"cmMotor"(Regime := "dbUnit".Unit[1].Regime, FQ := "dbMotors".M2_SPREDAJ_DESNO);
	"cmMotor"(Regime := "dbUnit".Unit[1].Regime, FQ := "dbMotors".M1_ZADAJ_LEVO);
	"cmMotor"(Regime := "dbUnit".Unit[1].Regime, FQ := "dbMotors".M2_SPREDAJ_LEVO);
	"cmMotor"(Regime := "dbUnit".Unit[1].Regime, FQ := "dbMotors".VKLOP_VIBRATORJA);
	"cmMotor"(Regime := "dbUnit".Unit[1].Regime, FQ := "dbMotors".VKLOP_M_TRAKA_VIJACNIKA);
	//----------------------------------------------------------------------
	//  write output
	"dbDO".VKLOP_M_TRACNEGA_TRANS_NOGIC := "dbMotors".VKLOP_M_TRACNEGA_TRANS_NOGIC.XS;
	
	"dbDO".MOTOR_1_ZADAJ_DESNO_START        := "dbMotors".M1_ZADAJ_DESNO.XS;
	"dbDO".MOTOR_1_ZADAJ_DESNO_HITROST      := "dbMotors".M1_ZADAJ_DESNO.Speed1Out;
	"dbDO".MOTOR_1_ZADAJ_DESNO_SMER         := "dbMotors".M1_ZADAJ_DESNO.Direction;
	
	"dbDO".MOTOR_2_SPREDAJ_DESNO_START      := "dbMotors".M2_SPREDAJ_DESNO.XS;
	"dbDO".MOTOR_2_SPREDAJ_DESNO_HITROST    := "dbMotors".M2_SPREDAJ_DESNO.Speed1Out;
	"dbDO".MOTOR_2_SPREDAJ_DESNO_SMER       := "dbMotors".M2_SPREDAJ_DESNO.Direction;
	
	"dbDO".MOTOR_1_ZADAJ_LEVO_START         := "dbMotors".M1_ZADAJ_LEVO.XS;
	"dbDO".MOTOR_1_ZADAJ_LEVO_HITROST       := "dbMotors".M1_ZADAJ_LEVO.Speed1Out;
	"dbDO".MOTOR_1_ZADAJ_LEVO_SMER          := "dbMotors".M1_ZADAJ_LEVO.Direction;
	
	"dbDO".MOTOR_2_SPREDAJ_LEVO_START       := "dbMotors".M2_SPREDAJ_LEVO.XS;
	"dbDO".MOTOR_2_SPREDAJ_LEVO_HITROST     := "dbMotors".M2_SPREDAJ_LEVO.Speed1Out;
	"dbDO".MOTOR_2_SPREDAJ_LEVO_SMER        := "dbMotors".M2_SPREDAJ_LEVO.Direction;
	
	"dbDO".VKLOP_VIBRATORJA := "dbMotors".VKLOP_VIBRATORJA.XS;
	"dbDO".VKLOP_M_TRAKA_VIJACNIKA := "dbMotors".VKLOP_M_TRAKA_VIJACNIKA.XS;
END_FUNCTION

FUNCTION "cmMotor" : Void
{ S7_Optimized_Access := 'TRUE' }
VERSION : 0.1
   VAR_IN_OUT 
      Regime : USInt;
      FQ : "udtMotor";
   END_VAR

   VAR_TEMP 
      tmpTimer : Int;
      tmpTimerDelay : Int;
   END_VAR

   VAR CONSTANT 
      FILTER_TIME_ResetFCAlarm : UInt := 10;
   END_VAR


BEGIN
	//HMI ovveride
	IF #FQ.ToggleCmd THEN
	    #FQ.ManON  := NOT #FQ.ManON;
	    #FQ.ManOFF := NOT #FQ.ManON;
	    #FQ.ToggleCmd := False;
	END_IF;
	
	//----------------------------------------------------------------------
	//  ALARMING MODULE
	IF #FQ.AlarmAck THEN
	    #FQ.AlarmEA := FALSE;
	    #FQ.AlarmESA := FALSE;
	    #FQ.AlarmFSL := FALSE;
	    #FQ.AlarmAck := FALSE;
	    #FQ.Alarm := FALSE;
	    #FQ.Timer_EA := 0;
	    #FQ.Timer_FSL := 0;
	    
	    #FQ.ResetFCAlarm := TRUE;
	END_IF;
	
	// Thermal overlload - ESA (0 = OK; 1 = ALARM)
	#FQ.AlarmESA := NOT #FQ.ESA;
	
	// Motor running - EA (0 = ALARM; 1 = OK)    
	IF (#FQ.XS AND NOT #FQ.EA) OR (NOT #FQ.XS AND #FQ.EA) THEN
	    IF (#FQ.Timer_EA < #FQ.FILTER_TIME_EA) AND "100msOSR" THEN
	        #FQ.Timer_EA := #FQ.Timer_EA + 1;
	    END_IF;
	    IF (#FQ.Timer_EA >= #FQ.FILTER_TIME_EA) THEN
	        #FQ.AlarmEA := TRUE;
	    END_IF;
	ELSE
	    #FQ.Timer_EA := 0;
	END_IF;
	
	// Flow Switch Sensor - FSL (0 = ALARM; 1 = OK)     
	IF (#FQ.XS AND #FQ.EA AND NOT #FQ.FSL) THEN
	    IF (#FQ.Timer_FSL < #FQ.FILTER_TIME_FSL) AND "100msOSR" THEN
	        #FQ.Timer_FSL := #FQ.Timer_FSL + 1;
	    END_IF;
	    IF (#FQ.Timer_FSL >= #FQ.FILTER_TIME_FSL) THEN
	        #FQ.AlarmFSL := TRUE;
	    END_IF;
	END_IF;
	
	IF (#FQ.XS AND #FQ.FSL) OR (NOT #FQ.XS) THEN
	    #FQ.Timer_FSL := 0;
	END_IF;
	
	IF #FQ.ResetFCAlarm THEN
	    IF (#FQ.Timer_ResetFCAlarm < #FILTER_TIME_ResetFCAlarm) AND "100msOSR" THEN // 1 sec
	        #FQ.Timer_ResetFCAlarm := #FQ.Timer_ResetFCAlarm + 1;
	    END_IF;
	    IF (#FQ.Timer_ResetFCAlarm >= #FILTER_TIME_ResetFCAlarm) THEN
	        #FQ.Timer_ResetFCAlarm := 0;
	        #FQ.ResetFCAlarm := FALSE;
	    END_IF;
	END_IF;
	
	//----------------------------------------------------------------------
	//  DIGITAL OUTPUT
	#FQ.XS := FALSE;
	#FQ.Speed1Out := FALSE;
	#FQ.Speed1Out := FALSE;
	
	IF (#Regime = 0) THEN
	    #FQ.ManON := FALSE;
	    #FQ.ManOFF := FALSE;
	    #FQ.XS := #FQ.AutoON;
	ELSIF (#Regime > 0) THEN
	    #FQ.XS := (#FQ.AutoON AND NOT #FQ.ManON AND NOT #FQ.ManOFF) OR (#FQ.ManON AND NOT #FQ.ManOFF);
	END_IF;
	
	//----------------------------------------------------------------------
	// ANALOG OUTPUT
	//select which source to use
	IF (#Regime = 0) THEN
	    #FQ.ManSpeed := -1.0;
	    #FQ.OutRPM := ((#FQ.MaxEng - #FQ.MinEng) * 100.0) / #FQ.AutoSpeed;
	    
	    #FQ.Speed1Out := (#FQ.AutoSpeed = 1.0);
	    #FQ.Speed2Out := (#FQ.AutoSpeed = 2.0);
	END_IF;
	
	IF (#Regime >= 1) THEN
	    IF (#FQ.ManSpeed <> -1.0) THEN
	        #FQ.OutRPM := ((#FQ.MaxEng - #FQ.MinEng) * 100.0) / #FQ.ManSpeed;
	        #FQ.Speed1Out := (#FQ.ManSpeed = 1.0);
	        #FQ.Speed2Out := (#FQ.ManSpeed = 2.0);
	    ELSE
	        #FQ.OutRPM := ((#FQ.MaxEng - #FQ.MinEng) * 100.0) / #FQ.AutoSpeed;
	        #FQ.Speed1Out := (#FQ.ManSpeed = 1.0);
	        #FQ.Speed2Out := (#FQ.ManSpeed = 2.0);
	    END_IF;
	END_IF;
	
	// check output
	IF (#FQ.OutRPM >= #FQ.MaxEng) THEN
	    #FQ.OutRPM := #FQ.MaxEng;
	END_IF;
	IF (#FQ.OutRPM <= #FQ.MinEng) THEN
	    #FQ.OutRPM := #FQ.MinEng;
	END_IF;
	
	// scale to % units
	#FQ.OutPrc := (#FQ.OutRPM / (#FQ.MaxEng - #FQ.MinEng)) * 100;
	IF #FQ.OutPrc < 0 THEN
	    #FQ.OutPrc := 0;
	ELSIF #FQ.OutPrc > 100 THEN
	    #FQ.OutPrc := 100;
	END_IF;
	
	//----------------------------------------------------------------------
	// manual
	#FQ.Manual := #FQ.ManON OR #FQ.ManOFF;
	
	//----------------------------------------------------------------------
	// FQ common failure (active, when one of the above alarms active)
	IF #FQ.AlarmEA OR #FQ.AlarmESA OR #FQ.AlarmFSL OR #FQ.Alarm THEN
	    #FQ.Alarm   := TRUE;
	    #FQ.AutoON  := FALSE;
	    #FQ.ManON   := FALSE;
	    #FQ.ManOFF  := FALSE;
	    #FQ.XS      := FALSE;
	    
	    //else
	    //  FQ.Alarm := FALSE;
	END_IF;
	//----------------------------------------------------------------------
	//  interlock
	IF #FQ.Interlock AND (#Regime < 2) THEN
	    #FQ.XS := FALSE;
	    #FQ.OutPrc := 0.0;
	    #FQ.OutRPM := 0.0;
	END_IF;
	
	//----------------------------------------------------------------------
	//  direction
	#FQ.Direction := #FQ.DirectionReq;
	
END_FUNCTION

FUNCTION "fcWriteOUT" : Void
{ S7_Optimized_Access := 'TRUE' }
VERSION : 0.1

BEGIN
	// Write DO output (14x) to CPU
	// Write outputs from DB11.DBB0 with 2 bytes to Q0.0-Q1.0 
	POKE_BLK(area_src := 16#84, // DB
	         dbNumber_src := 11,
	         byteOffset_src := 0,
	         area_dest := 16#82, // PQ
	         dbNumber_dest := 0,
	         byteOffset_dest := 0,
	         count := 2);
	
	// Write DO output (16x2) to Weidmuller UR20-FBC-PN-IRT-V2
	// Write outputs from DB11.DBB2 with 4 bytes to Q2.0-Q5.0
	POKE_BLK(area_src := 16#84, // DB
	         dbNumber_src := 11,
	         byteOffset_src := 2,
	         area_dest := 16#82, // PQ
	         dbNumber_dest := 0,
	         byteOffset_dest := 2,
	         count := 4);
	
	// Write PDO output (32) to SMC_EX260-S1
	// Write outputs from DB12.DBB0 with 4 bytes to Q6.0-Q9.0 
	POKE_BLK(area_src := 16#84, // DB
	         dbNumber_src := 12,
	         byteOffset_src := 0,
	         area_dest := 16#82, // PQ
	         dbNumber_dest := 0,
	         byteOffset_dest := 6,
	         count := 4);
	
END_FUNCTION

ORGANIZATION_BLOCK "Cyclic interrupt"   // OB35, LAD, CyclicInterrupt
{ S7_Optimized_Access := 'TRUE' }
VERSION : 0.1
// stored: AutoNumber false, IsIECCheckEnabled false, SetENOAutomatically false
   VAR_INPUT
      Initial_Call : Bool;   // Initial call of this OB
      Event_Count : Int;   // Events discarded
   END_VAR
   VAR_TEMP
      OB35_EV_CLASS : Byte;   // Bits 0-3 = 1 (Coming event), Bits 4-7 = 1 (Event class 1)
      OB35_STRT_INF : Byte;   // 16#36 (OB 35 has started)
      OB35_PRIORITY : Byte;   // Priority of OB Execution
      OB35_OB_NUMBR : Byte;   // 35 (Organization block 35, OB35)
      OB35_RESERVED_1 : Byte;   // Reserved for system
      OB35_RESERVED_2 : Byte;   // Reserved for system
      OB35_PHASE_OFFSET : Word;   // Phase offset (msec)
      OB35_RESERVED_3 : Int;   // Reserved for system
      OB35_EXC_FREQ : Int;   // Frequency of execution (msec)
      OB35_DATE_TIME : DTL;   // Date and time OB35 started
   END_VAR
BEGIN
END_ORGANIZATION_BLOCK

ORGANIZATION_BLOCK "Diagnostic error interrupt"   // OB82, LAD, DiagnosticErrorInterrupt
{ S7_Optimized_Access := 'TRUE' }
VERSION : 0.1
// stored: IsIECCheckEnabled false, SetENOAutomatically false
   VAR_INPUT
      IO_State : Word;   // IO state of the HW object
      LADDR : HW_ANY;   // Hardware identifier
      Channel : UInt;   // Channel number
      MultiError : Bool;   // =true if more than one error is present
   END_VAR
BEGIN
END_ORGANIZATION_BLOCK

ORGANIZATION_BLOCK "Profile"   // OB57, LAD, Profile
TITLE = "DP:manufacture_alarm"
{ S7_Optimized_Access := 'TRUE' }
VERSION : 0.1
// stored: IsIECCheckEnabled false, SetENOAutomatically false
   VAR_INPUT
      LADDR : HW_IO;   // Hardware identifier
      Slot : UInt;   // Slot number
      Specifier : Word;   // alarm specifier out of the alarm telegram
   END_VAR
BEGIN
END_ORGANIZATION_BLOCK

ORGANIZATION_BLOCK "Pull or plug of modules"   // OB83, LAD, PullOrPlugOfModules
{ S7_Optimized_Access := 'TRUE' }
VERSION : 0.1
// stored: IsIECCheckEnabled false, SetENOAutomatically false
   VAR_INPUT
      LADDR : HW_IO;   // Hardware identifier
      Event_Class : Byte;   // 16#38/39: module inserted, removed
      Fault_ID : Byte;   // Fault identifier
   END_VAR
BEGIN
END_ORGANIZATION_BLOCK

ORGANIZATION_BLOCK "Rack or station failure"   // OB86, LAD, RackOrStationFailure
{ S7_Optimized_Access := 'TRUE' }
VERSION : 0.1
// stored: IsIECCheckEnabled false, SetENOAutomatically false
   VAR_INPUT
      LADDR : HW_DEVICE;   // Hardware identifier
      Event_Class : Byte;   // Event class
      Fault_ID : Byte;   // Fault identifier
   END_VAR
BEGIN
END_ORGANIZATION_BLOCK

ORGANIZATION_BLOCK "Startup"   // OB100, LAD, Startup
TITLE = "Complete Restart"
{ S7_Optimized_Access := 'TRUE' }
VERSION : 0.1
// stored: AutoNumber true, IsIECCheckEnabled false, SetENOAutomatically false
   VAR_INPUT
      LostRetentive : Bool;   // True if retentive data are lost
      LostRTC : Bool;   // True if date and time are lost
   END_VAR
BEGIN

REGION Network 1
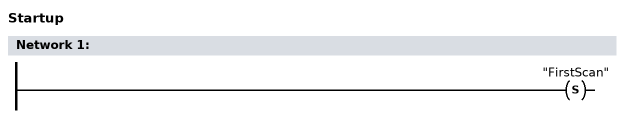
   RUNG wire#powerrail
      S_Coil( "FirstScan" )
   END_RUNG
   // the same network as SCL:
   "FirstScan" := TRUE;
END_REGION
END_ORGANIZATION_BLOCK

ORGANIZATION_BLOCK "Status"   // OB55, LAD, Status
TITLE = "DP:status_alarm"
{ S7_Optimized_Access := 'TRUE' }
VERSION : 0.1
// stored: IsIECCheckEnabled false, SetENOAutomatically false
   VAR_INPUT
      LADDR : HW_IO;   // Hardware identifier
      Slot : UInt;   // Slot number
      Specifier : Word;   // alarm specifier out of the alarm telegram
   END_VAR
BEGIN
END_ORGANIZATION_BLOCK

ORGANIZATION_BLOCK "Time error interrupt"   // OB80, LAD, TimeErrorInterrupt
{ S7_Optimized_Access := 'TRUE' }
VERSION : 0.1
// stored: IsIECCheckEnabled false, SetENOAutomatically false
   VAR_INPUT
      Fault_ID : Byte;   // Fault identifier
      Csg_OBnr : OB_ANY;   // Number of OB causing the error
      Csg_Prio : UInt;   // Priority of OB causing the error
   END_VAR
BEGIN
END_ORGANIZATION_BLOCK

ORGANIZATION_BLOCK "Update"   // OB56, LAD, Update
TITLE = "DP:update_alarm"
{ S7_Optimized_Access := 'TRUE' }
VERSION : 0.1
// stored: IsIECCheckEnabled false, SetENOAutomatically false
   VAR_INPUT
      LADDR : HW_IO;   // Hardware identifier
      Slot : UInt;   // Slot number
      Specifier : Word;   // alarm specifier out of the alarm telegram
   END_VAR
BEGIN
END_ORGANIZATION_BLOCK

FUNCTION "cmFindStrgEQ" : Bool   // FC220, LAD
{ S7_Optimized_Access := 'TRUE' }
VERSION : 0.1
// stored: AutoNumber false, IsIECCheckEnabled false, SetENOAutomatically false, UDAEnableTagReadback false
   VAR_INPUT
      String1 : String;
      String2 : String;
   END_VAR
BEGIN

REGION Network 1
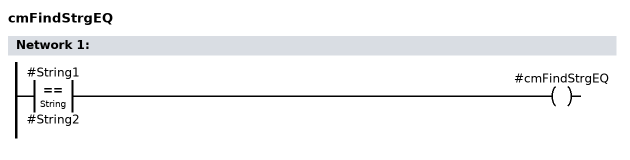
   RUNG wire#powerrail
      { S7_Templates := "SrcType := String" } EQ_Contact(in1 := #String1, in2 := #String2)
      Coil( #cmFindStrgEQ )
   END_RUNG
   // the same network as SCL:
   #cmFindStrgEQ := #String1 = #String2;
END_REGION
END_FUNCTION

FUNCTION "BIT_SET_WORD" : Void
{ S7_Optimized_Access := 'FALSE' }
VERSION : 0.1
   VAR_INPUT 
      Value : Bool;
      No_Bit : Int;
   END_VAR

   VAR_IN_OUT 
      In_Out_Word : Word;
   END_VAR

   VAR_TEMP 
      Input_Word_Temp_1 : Word;
      Input_Word_Temp_2 : Word;
   END_VAR


BEGIN
	IF #Value THEN
	    #Input_Word_Temp_1 := 2#0000_0000_0000_0001;
	ELSE
	    #Input_Word_Temp_1 := 2#0000_0000_0000_0000;
	END_IF;
	
	#Input_Word_Temp_2 := #In_Out_Word;
	
	IF SHR(IN := #Input_Word_Temp_2, N := #No_Bit - 1) = 0 THEN
	    #Input_Word_Temp_1 := SHL(IN := #Input_Word_Temp_1, N := #No_Bit - 1);
	    #In_Out_Word := INT_TO_WORD(WORD_TO_INT(#Input_Word_Temp_2) + WORD_TO_INT(#Input_Word_Temp_1));
	ELSE
	    #In_Out_Word := #In_Out_Word;
	END_IF;
	
END_FUNCTION

FUNCTION_BLOCK "op_ButtonHelix_3"
{ S7_Optimized_Access := 'TRUE' }
VERSION : 0.1
   VAR_IN_OUT 
      SEMAFOR_ZELENA : "udtDigitalValve";
      SEMAFOR_RUMENA : "udtDigitalValve";
      SEMAFOR_RDECA : "udtDigitalValve";
      VKLOP_VIBRATORJA : "udtMotor";
      VKLOP_M_TRACNEGA_TRANS_NOGIC : "udtMotor";
   END_VAR

   VAR RETAIN
      CurrentStep { ExternalAccessible := 'False'; ExternalVisible := 'False'; ExternalWritable := 'False'} : Int;
      PhaseStatus { ExternalAccessible := 'False'; ExternalVisible := 'False'; ExternalWritable := 'False'} : Int;   // // 0=IDLE, 5=RUNNING, 6=HOLD
      AlarmPresent { ExternalAccessible := 'False'; ExternalVisible := 'False'; ExternalWritable := 'False'} : Bool;
      InitPosition { ExternalAccessible := 'False'; ExternalVisible := 'False'; ExternalWritable := 'False'} : Bool;
   END_VAR
   VAR 
      IEC_TimerOnDly_1 {InstructionName := 'TONR_TIME'; LibVersion := '1.0'; ExternalAccessible := 'False'; ExternalVisible := 'False'; ExternalWritable := 'False'; S7_SetPoint := 'False'} : TONR_TIME;
      IEC_TimerOnDly_2 {InstructionName := 'TONR_TIME'; LibVersion := '1.0'; ExternalAccessible := 'False'; ExternalVisible := 'False'; ExternalWritable := 'False'; S7_SetPoint := 'False'} : TONR_TIME;
      IEC_TimerOnDly_3 {InstructionName := 'TONR_TIME'; LibVersion := '1.0'; ExternalAccessible := 'False'; ExternalVisible := 'False'; ExternalWritable := 'False'; S7_SetPoint := 'False'} : TONR_TIME;
      IEC_TimerOnDly_4 {InstructionName := 'TONR_TIME'; LibVersion := '1.0'; ExternalAccessible := 'False'; ExternalVisible := 'False'; ExternalWritable := 'False'; S7_SetPoint := 'False'} : TONR_TIME;
      IEC_TimerOnDly_5 {InstructionName := 'TONR_TIME'; LibVersion := '1.0'; ExternalAccessible := 'False'; ExternalVisible := 'False'; ExternalWritable := 'False'; S7_SetPoint := 'False'} : TONR_TIME;
      IEC_TimerOnDly_6 {InstructionName := 'TONR_TIME'; LibVersion := '1.0'; ExternalAccessible := 'False'; ExternalVisible := 'False'; ExternalWritable := 'False'; S7_SetPoint := 'False'} : TONR_TIME;
      IEC_TimerOnDly_7 {InstructionName := 'TONR_TIME'; LibVersion := '1.0'; ExternalAccessible := 'False'; ExternalVisible := 'False'; ExternalWritable := 'False'; S7_SetPoint := 'False'} : TONR_TIME;
      IEC_TimerOnDly_8 {InstructionName := 'TONR_TIME'; LibVersion := '1.0'; ExternalAccessible := 'False'; ExternalVisible := 'False'; ExternalWritable := 'False'; S7_SetPoint := 'False'} : TONR_TIME;
      IEC_TimerOnDly_9 {InstructionName := 'TONR_TIME'; LibVersion := '1.0'; ExternalAccessible := 'False'; ExternalVisible := 'False'; ExternalWritable := 'False'; S7_SetPoint := 'False'} : TONR_TIME;
      IEC_TimerOnDly_10 {InstructionName := 'TONR_TIME'; LibVersion := '1.0'; ExternalAccessible := 'False'; ExternalVisible := 'False'; ExternalWritable := 'False'; S7_SetPoint := 'False'} : TONR_TIME;
      IEC_TimerOnDly_ET_1 { ExternalAccessible := 'False'; ExternalVisible := 'False'; ExternalWritable := 'False'} : Time;
      IEC_TimerOnDly_ET_2 { ExternalAccessible := 'False'; ExternalVisible := 'False'; ExternalWritable := 'False'} : Time;
      IEC_TimerOnDly_ET_3 { ExternalAccessible := 'False'; ExternalVisible := 'False'; ExternalWritable := 'False'} : Time;
      IEC_TimerOnDly_ET_4 { ExternalAccessible := 'False'; ExternalVisible := 'False'; ExternalWritable := 'False'} : Time;
      IEC_TimerOnDly_ET_5 { ExternalAccessible := 'False'; ExternalVisible := 'False'; ExternalWritable := 'False'} : Time;
      IEC_TimerOnDly_ET_6 { ExternalAccessible := 'False'; ExternalVisible := 'False'; ExternalWritable := 'False'} : Time;
      IEC_TimerOnDly_ET_7 { ExternalAccessible := 'False'; ExternalVisible := 'False'; ExternalWritable := 'False'} : Time;
      IEC_TimerOnDly_ET_8 { ExternalAccessible := 'False'; ExternalVisible := 'False'; ExternalWritable := 'False'} : Time;
      IEC_TimerOnDly_ET_9 { ExternalAccessible := 'False'; ExternalVisible := 'False'; ExternalWritable := 'False'} : Time;
      IEC_TimerOnDly_ET_10 { ExternalAccessible := 'False'; ExternalVisible := 'False'; ExternalWritable := 'False'} : Time;
      IEC_TimerOnDly_DN_1 { ExternalAccessible := 'False'; ExternalVisible := 'False'; ExternalWritable := 'False'} : Bool;
      IEC_TimerOnDly_DN_2 { ExternalAccessible := 'False'; ExternalVisible := 'False'; ExternalWritable := 'False'} : Bool;
      IEC_TimerOnDly_DN_3 { ExternalAccessible := 'False'; ExternalVisible := 'False'; ExternalWritable := 'False'} : Bool;
      IEC_TimerOnDly_DN_4 { ExternalAccessible := 'False'; ExternalVisible := 'False'; ExternalWritable := 'False'} : Bool;
      IEC_TimerOnDly_DN_5 { ExternalAccessible := 'False'; ExternalVisible := 'False'; ExternalWritable := 'False'} : Bool;
      IEC_TimerOnDly_DN_6 { ExternalAccessible := 'False'; ExternalVisible := 'False'; ExternalWritable := 'False'} : Bool;
      IEC_TimerOnDly_DN_7 { ExternalAccessible := 'False'; ExternalVisible := 'False'; ExternalWritable := 'False'} : Bool;
      IEC_TimerOnDly_DN_8 { ExternalAccessible := 'False'; ExternalVisible := 'False'; ExternalWritable := 'False'} : Bool;
      IEC_TimerOnDly_DN_9 { ExternalAccessible := 'False'; ExternalVisible := 'False'; ExternalWritable := 'False'} : Bool;
      IEC_TimerOnDly_DN_10 { ExternalAccessible := 'False'; ExternalVisible := 'False'; ExternalWritable := 'False'} : Bool;
      Mode : Int;
      ModePrev : Int;
   END_VAR
   VAR RETAIN
      CurrUserN_LEN : Int;
   END_VAR
   VAR 
      HMICurrScreenOLD : Byte;
      AlarmPresentOLD { ExternalAccessible := 'False'; ExternalVisible := 'False'; ExternalWritable := 'False'} : Bool;
      InitPositionOLD { ExternalAccessible := 'False'; ExternalVisible := 'False'; ExternalWritable := 'False'} : Bool;
   END_VAR
   VAR RETAIN
      DlyTimeToStart_TRAK_VIJAC { ExternalAccessible := 'False'; ExternalVisible := 'False'; ExternalWritable := 'False'; S7_SetPoint := 'True'} : Int := 7;
      DlyTimeToStop_TRAK_VIJAC { ExternalAccessible := 'False'; ExternalVisible := 'False'; ExternalWritable := 'False'; S7_SetPoint := 'True'} : Int := 20;
      DlyTimeToStart_VIBRO { ExternalAccessible := 'False'; ExternalVisible := 'False'; ExternalWritable := 'False'; S7_SetPoint := 'True'} : Int := 30;
      DlyTimeToStop_VIBRO { ExternalAccessible := 'False'; ExternalVisible := 'False'; ExternalWritable := 'False'; S7_SetPoint := 'True'} : Int := 10;
   END_VAR
   VAR 
      UnitRegimeOLD { ExternalAccessible := 'False'; ExternalVisible := 'False'; ExternalWritable := 'False'} : Int;
      EndTransportNogic { ExternalAccessible := 'False'; ExternalVisible := 'False'; ExternalWritable := 'False'} : Bool;
      Count_M_TRACNEGA_TRANS_NOGIC { ExternalAccessible := 'False'; ExternalVisible := 'False'; ExternalWritable := 'False'} : USInt;
   END_VAR
   VAR RETAIN
      DlyTimeForAlarmAddNewHelix { ExternalAccessible := 'False'; ExternalVisible := 'False'; ExternalWritable := 'False'} : UInt;
   END_VAR
   VAR 
      Count_M_TRACNEGA_TRANS_NOGIC_OLD { ExternalAccessible := 'False'; ExternalVisible := 'False'; ExternalWritable := 'False'} : USInt;
   END_VAR

   VAR_TEMP 
      i : Int;
      j : Int;
      i1 : Int;
      i2 : Int;
      i3 : Int;
      i4 : Int;
      i5 : Int;
      i6 : Int;
      i7 : Int;
      i8 : Int;
      i9 : Int;
      i10 : Int;
   END_VAR

   VAR CONSTANT 
      PLIIndex : Int := 3;
   END_VAR


BEGIN
	// Initialize variables
	#i := 0;
	#j := 0;
	#CurrUserN_LEN      := LEN("dbHMIUser".CurrentUsername); // if 0 user not logged IN, if > 0 user is logged IN
	
	#i1   := #PLIIndex;                          // 1
	#i2   := #PLIIndex + "MaxPLITimersIndex";    // 5
	#i3   := #PLIIndex + 2*"MaxPLITimersIndex";  // 9
	#i4   := #PLIIndex + 3*"MaxPLITimersIndex";  // 13
	#i5   := #PLIIndex + 4*"MaxPLITimersIndex";  // 17
	#i6   := #PLIIndex + 5*"MaxPLITimersIndex";  // 21
	#i7   := #PLIIndex + 6*"MaxPLITimersIndex";  // 25
	#i8   := #PLIIndex + 7*"MaxPLITimersIndex";  // 29
	#i9   := #PLIIndex + 8*"MaxPLITimersIndex";  // 33
	#i10  := #PLIIndex + 9*"MaxPLITimersIndex";  // 37
	
	// Check alarms
	#AlarmPresent := 0;
	// 20210517_PRA FOR #i := 1 TO 32 DO Alarm [8] is a warning and light on YELOW light, not red light as others PLI alarms (see fcUtilities)
	FOR #i := 1 TO 7 DO
	  IF "dbAlarms".PLI[#PLIIndex, #i] THEN
	    #AlarmPresent := 1;
	  END_IF;
	  IF "AlarmAck" THEN
	    "dbAlarms".PLI[#PLIIndex, #i] := 0;
	  END_IF;
	END_FOR;
	
	// Timers section
	#IEC_TimerOnDly_DN_1 := 0;
	#IEC_TimerOnDly_1(IN := False,
	                  R := False,
	                  PT := T#10s,
	                  Q => #IEC_TimerOnDly_DN_1,
	                  ET => #IEC_TimerOnDly_ET_1);
	
	(*
	// Alarms reset timer
	#IEC_TimerOnDly_4_DN := 0;
	#IEC_TimerOnDly_4(IN := "HS_RESET",
	                  R := NOT "HS_RESET",
	                  PT := T#2s,
	                  Q => #IEC_TimerOnDly_4_DN,
	                  ET => #IEC_TimerOnDly_4_ET);
	IF "HS_RESET" THEN
	    "dbDigitalValves".XS_FC_RESET.AutoON := true;
	END_IF;
	*)
	
	// PHASE STATUS
	#PhaseStatus := 0;
	IF #CurrentStep >= 1 AND "dbUnit".Unit[1].StartStop THEN
	  #PhaseStatus := 5;
	END_IF;
	IF #CurrentStep >= 1 AND (NOT "dbUnit".Unit[1].StartStop OR NOT "dbDigitalSensors".ZAUSTAVITEV_V_SILI_NI_AKTIVIRANA.InputF) THEN
	  #CurrentStep := 0; // // Operation is stopped
	  #PhaseStatus := 7;
	END_IF;
	IF #CurrentStep >= 1 AND #AlarmPresent THEN
	  #PhaseStatus := 6;
	END_IF;
	
	// Stop unit if regime is changed
	IF "dbUnit".Unit[1].Regime <> #UnitRegimeOLD THEN
	  "dbUnit".Unit[1].StartStop := False;
	END_IF;
	
	CASE #CurrentStep OF
	  0: // Sequence permissives
	    // STOP phases
	    "ph_Helix_1_DB".#StartCmd         := False;
	    "ph_LegsShifter_2_DB".#StartCmd   := False;
	
	    "dbHMIUser".CurrMachineStep := 'Pritisni START';
	
	    IF ("dbUnit".Unit[1].Regime=0 AND "dbUnit".Unit[1].StartStop) THEN // Local  mode
	      IF #PhaseStatus=0 THEN
	        "dbHMIUser".CurrMachineStep := 'Zagon naprave v teku';
	        #CurrentStep := 3;
	      END_IF;
	    END_IF;
	
	  3: // Check initial positions
	    "dbHMIUser".CurrMachineStep := 'Naprava v alarmu';
	
	    IF NOT "dbUnit".Unit[1].AlarmsPresent THEN
	      #CurrentStep := 5;
	    END_IF;
	
	  5: // Init variables
	    "dbTimers".Num[#i1].EE    := False;
	    "dbTimers".Num[#i2].EE    := False;
	    "dbTimers".Num[#i3].EE    := False;
	    "dbTimers".Num[#i4].EE    := False;
	    "dbTimers".Num[#i5].EE    := False;
	    "dbTimers".Num[#i6].EE    := False;
	    "dbTimers".Num[#i7].EE    := False;
	    "dbTimers".Num[#i8].EE    := False;
	    "dbTimers".Num[#i9].EE    := False;
	    "dbTimers".Num[#i10].EE   := False;
	
	    #EndTransportNogic := False;
	    #Count_M_TRACNEGA_TRANS_NOGIC := 0;
	    #Count_M_TRACNEGA_TRANS_NOGIC_OLD := #Count_M_TRACNEGA_TRANS_NOGIC;
	    
	    // "ph_LegsShifter_2_DB"."Mode" := 1; // Start fill slide LEVO, then start fill slide DESNO to the top
	    "dbHMIUser".CurrMachineStep := 'Transport nogic do vijacnega dela v teku';
	
	    #CurrentStep := 10;
	
	  10: // Move legs with VKLOP_M_TRAKA_VIJACNIKA to VIBRATOR
	    "ph_Helix_1_DB".#StartCmd         := True;
	    IF ("ph_Helix_1_DB".CurrentStep>5) THEN // Wait to run #VKLOP_M_TRAKA_VIJACNIKA till legs reach TRAK_LEVO1, TRAK_LEVO2, TRAK_DESNO1, TRAK_DESNO2 
	      "ph_LegsShifter_2_DB".#StartCmd := True;
	    END_IF;
	
	// START/STOP TRAKA_VIJACNIKA
	REGION START/STOP TRAKA ZA TRANSPORT NOGIC V VIBRATOR
	    // "dbDigitalSensors".NOGICE_V_VIBRATORJU.InputF=1 nogice niso prisotne
	    // 20210512_PRA "dbTimers".Num[#i1].EE  := "dbDigitalSensors".NOGICE_V_VIBRATORJU.InputF;
	    "dbTimers".Num[#i1].EE  := "dbDigitalSensors".NOGICE_V_VIBRATORJU.InputF;
	    "dbTimers".Num[#i1].PRE := #DlyTimeToStart_TRAK_VIJAC;
	
	    IF ("dbTimers".Num[#i1].EE AND "dbTimers".Num[#i1].DN) OR "dbTimers".Num[#i2].TT THEN
	      #VKLOP_M_TRACNEGA_TRANS_NOGIC.AutoON := True; // Start, če ni prisotnih nogic v vibratorju in iztek časovnika. Stop po preteku časa ali prisotnosti nogic v vibratorju.
	      "dbTimers".Num[#i2].EE  := True;
	      "dbTimers".Num[#i2].PRE := #DlyTimeToStop_TRAK_VIJAC;
	    END_IF;
	    IF "dbTimers".Num[#i2].EE AND "dbTimers".Num[#i2].DN THEN
	      "dbTimers".Num[#i2].EE  := False;
	      "dbTimers".Num[#i2].DN  := False;
	
	      #EndTransportNogic := True;
	      "dbTimers".Num[#i1].ACC  := 0;
	      #Count_M_TRACNEGA_TRANS_NOGIC := #Count_M_TRACNEGA_TRANS_NOGIC + 1;
	    END_IF;
	  
	    IF (#Count_M_TRACNEGA_TRANS_NOGIC_OLD <> #Count_M_TRACNEGA_TRANS_NOGIC) THEN
	        #Count_M_TRACNEGA_TRANS_NOGIC := #Count_M_TRACNEGA_TRANS_NOGIC + 1;
	    END_IF;
	    #Count_M_TRACNEGA_TRANS_NOGIC_OLD := #Count_M_TRACNEGA_TRANS_NOGIC;
	END_REGION
	
	REGION START/STOP VIBRATORJA
	    // 20210512_PRA "dbTimers".Num[#i3].EE  := NOT "dbDigitalSensors".FOTOCELICA_VSTOP_DRCA_NOGIC.InputF;
	    "dbTimers".Num[#i3].EE  := NOT "dbDigitalSensors".FOTOCELICA_VSTOP_DRCA_NOGIC.InputF OR #EndTransportNogic;
	    "dbTimers".Num[#i3].PRE := #DlyTimeToStart_VIBRO;
	
	    IF ("dbTimers".Num[#i3].EE AND "dbTimers".Num[#i3].DN) OR "dbTimers".Num[#i4].TT THEN // zakasnitev delovanja
	      #VKLOP_VIBRATORJA.AutoON := True;
	
	      "dbTimers".Num[#i4].EE  := True;
	      "dbTimers".Num[#i4].PRE := #DlyTimeToStop_VIBRO;
	    END_IF;
	    IF "dbTimers".Num[#i4].EE AND "dbTimers".Num[#i4].DN THEN // zakasnitev mirovanja
	      "dbTimers".Num[#i4].EE  := False;
	      "dbTimers".Num[#i4].DN  := False;
	      #EndTransportNogic := False;
	
	      "dbTimers".Num[#i3].ACC  := 0; 
	    END_IF;
	END_REGION
	
	END_CASE;
	
	// ALARMS SECTION
	// Alarm 1
	// ZAUSTAVITEV_V_SILI_NI_AKTIVIRANA
	IF ("dbSystemAlarms".SysAlm[01]) THEN
	  "dbAlarms".PLI[#PLIIndex, 1] := 1;
	END_IF;
	
	// Alarm 2
	// PRISOTNOST_ZRAKA_NA_NAPRAVI
	IF ("dbSystemAlarms".SysAlm[02]) THEN
	  "dbAlarms".PLI[#PLIIndex, 2] := 1;
	END_IF;
	
	// Alarm 3
	// FOTO_ZAVESA_KANAL_1
	IF ("dbSystemAlarms".SysAlm[03]) THEN
	  ; // "dbAlarms".PLI[#PLIIndex, 3] := 1;
	END_IF;
	
	// Alarm 4
	// FOTO_ZAVESA_KANAL_2
	IF ("dbSystemAlarms".SysAlm[04]) THEN
	  ; // "dbAlarms".PLI[#PLIIndex, 4] := 1;
	END_IF;
	
	// Alarm 5
	IF (#VKLOP_M_TRACNEGA_TRANS_NOGIC.Alarm) THEN
	  "dbAlarms".PLI[#PLIIndex, 5] := 1;
	END_IF;
	
	// Alarm 6
	IF (#VKLOP_VIBRATORJA.Alarm) THEN
	  "dbAlarms".PLI[#PLIIndex, 6] := 1;
	END_IF;
	
	// Alarm 7
	// Prisoten eden od alarmov
	IF (#CurrentStep = 3) AND ("dbUnit".Unit[1].AlarmsPresent) THEN
	  "dbAlarms".PLI[#PLIIndex, 7] := 1;
	END_IF;
	
	// Warning 8 - Show yellow light - see fcUtilities
	// Dodaj nogice v vstopni zalogovnik - 3x(#Count_M_TRACNEGA_TRANS_NOGIC=7) ponovi trak transport in začne teči alarm timer
	"dbTimers".Num[#i5].EE  := NOT "dbDigitalSensors".FOTOCELICA_TRANSPORTA_NOGIC.InputF AND #Count_M_TRACNEGA_TRANS_NOGIC>=6 AND #DlyTimeForAlarmAddNewHelix>0;
	"dbTimers".Num[#i5].PRE := #DlyTimeForAlarmAddNewHelix;
	IF (#CurrentStep = 10) AND ("dbTimers".Num[#i5].EE AND "dbTimers".Num[#i5].DN) THEN
	  #Count_M_TRACNEGA_TRANS_NOGIC := 0;
	  "dbTimers".Num[#i5].EE := False;
	  "dbAlarms".PLI[#PLIIndex, 8] := 1;
	END_IF;
	
	
	// Alarms in running state
	IF #PhaseStatus = 5 THEN
	  // Alarms action
	  IF (NOT #AlarmPresentOLD AND #AlarmPresent) OR (NOT #InitPositionOLD AND #InitPosition) THEN
	    ; // #CurrentStep := 6;
	  END_IF;
	END_IF;
	
	// OLD SCAN
	#AlarmPresentOLD        := #AlarmPresent;
	#InitPositionOLD        := #InitPosition;
	#HMICurrScreenOLD       := "dbHMIUser".HMICurrScreen;
	#UnitRegimeOLD          := "dbUnit".Unit[1].Regime;
END_FUNCTION_BLOCK

FUNCTION_BLOCK "ph_Helix_1"
{ S7_Optimized_Access := 'TRUE' }
VERSION : 0.1
   VAR_IN_OUT 
      Y8_VijaLocev_Des : "udtDigitalValve";
      Y9_VijaStop_DesZad : "udtDigitalValve";
      Y2_VijaDesZad_Dvig : "udtDigitalValve";
      Y10_Centri_DesZad : "udtDigitalValve";
      Y3_VijaDesSpr_Dvig : "udtDigitalValve";
      Y11_Centri_DesSpr : "udtDigitalValve";
      Y12_VijaLocev_Lev : "udtDigitalValve";
      Y13_VijaStop_LevZad : "udtDigitalValve";
      Y4_VijaLevZad_Dvig : "udtDigitalValve";
      Y14_Centri_LevZad : "udtDigitalValve";
      Y5_VijaLevSpr_Dvig : "udtDigitalValve";
      Y15_Centri_LevSpr : "udtDigitalValve";
      Y16_VpenjanjeDna : "udtDigitalValve";
      M1_ZADAJ_LEVO : "udtMotor";
      M2_SPREDAJ_LEVO : "udtMotor";
      M1_ZADAJ_DESNO : "udtMotor";
      M2_SPREDAJ_DESNO : "udtMotor";
      VKLOP_M_TRAKA_VIJACNIKA : "udtMotor";
   END_VAR

   VAR RETAIN
      CurrentStep { ExternalAccessible := 'False'; ExternalVisible := 'False'; ExternalWritable := 'False'} : Int;
      PhaseStatus { ExternalAccessible := 'False'; ExternalVisible := 'False'; ExternalWritable := 'False'} : Int;   // // 0=IDLE, 5=RUNNING, 6=HOLD
   END_VAR
   VAR 
      AlarmPresent { ExternalAccessible := 'False'; ExternalVisible := 'False'; ExternalWritable := 'False'} : Bool;
      InitPosition { ExternalAccessible := 'False'; ExternalVisible := 'False'; ExternalWritable := 'False'} : Bool;
      StartCmd { ExternalAccessible := 'False'; ExternalVisible := 'False'; ExternalWritable := 'False'} : Bool;
      AlarmPresentOLD { ExternalAccessible := 'False'; ExternalVisible := 'False'; ExternalWritable := 'False'} : Bool;
      InitPositionOLD { ExternalAccessible := 'False'; ExternalVisible := 'False'; ExternalWritable := 'False'} : Bool;
      IEC_TimerOnDly_1 {InstructionName := 'TONR_TIME'; LibVersion := '1.0'; ExternalAccessible := 'False'; ExternalVisible := 'False'; ExternalWritable := 'False'; S7_SetPoint := 'False'} : TONR_TIME;
      IEC_TimerOnDly_2 {InstructionName := 'TONR_TIME'; LibVersion := '1.0'; ExternalAccessible := 'False'; ExternalVisible := 'False'; ExternalWritable := 'False'; S7_SetPoint := 'False'} : TONR_TIME;
      IEC_TimerOnDly_3 {InstructionName := 'TONR_TIME'; LibVersion := '1.0'; ExternalAccessible := 'False'; ExternalVisible := 'False'; ExternalWritable := 'False'; S7_SetPoint := 'False'} : TONR_TIME;
      IEC_TimerOnDly_4 {InstructionName := 'TONR_TIME'; LibVersion := '1.0'; ExternalAccessible := 'False'; ExternalVisible := 'False'; ExternalWritable := 'False'; S7_SetPoint := 'False'} : TONR_TIME;
      IEC_TimerOnDly_5 {InstructionName := 'TONR_TIME'; LibVersion := '1.0'; ExternalAccessible := 'False'; ExternalVisible := 'False'; ExternalWritable := 'False'; S7_SetPoint := 'False'} : TONR_TIME;
      IEC_TimerOnDly_6 {InstructionName := 'TONR_TIME'; LibVersion := '1.0'; ExternalAccessible := 'False'; ExternalVisible := 'False'; ExternalWritable := 'False'; S7_SetPoint := 'False'} : TONR_TIME;
      IEC_TimerOnDly_7 {InstructionName := 'TONR_TIME'; LibVersion := '1.0'; ExternalAccessible := 'False'; ExternalVisible := 'False'; ExternalWritable := 'False'; S7_SetPoint := 'False'} : TONR_TIME;
      IEC_TimerOnDly_8 {InstructionName := 'TONR_TIME'; LibVersion := '1.0'; ExternalAccessible := 'False'; ExternalVisible := 'False'; ExternalWritable := 'False'; S7_SetPoint := 'False'} : TONR_TIME;
      IEC_TimerOnDly_9 {InstructionName := 'TONR_TIME'; LibVersion := '1.0'; ExternalAccessible := 'False'; ExternalVisible := 'False'; ExternalWritable := 'False'; S7_SetPoint := 'False'} : TONR_TIME;
      IEC_TimerOnDly_10 {InstructionName := 'TONR_TIME'; LibVersion := '1.0'; ExternalAccessible := 'False'; ExternalVisible := 'False'; ExternalWritable := 'False'; S7_SetPoint := 'False'} : TONR_TIME;
      IEC_TimerOnDly_ET_1 { ExternalAccessible := 'False'; ExternalVisible := 'False'; ExternalWritable := 'False'} : Time;
      IEC_TimerOnDly_ET_2 { ExternalAccessible := 'False'; ExternalVisible := 'False'; ExternalWritable := 'False'} : Time;
      IEC_TimerOnDly_ET_3 { ExternalAccessible := 'False'; ExternalVisible := 'False'; ExternalWritable := 'False'} : Time;
      IEC_TimerOnDly_ET_4 { ExternalAccessible := 'False'; ExternalVisible := 'False'; ExternalWritable := 'False'} : Time;
      IEC_TimerOnDly_ET_5 { ExternalAccessible := 'False'; ExternalVisible := 'False'; ExternalWritable := 'False'} : Time;
      IEC_TimerOnDly_ET_6 { ExternalAccessible := 'False'; ExternalVisible := 'False'; ExternalWritable := 'False'} : Time;
      IEC_TimerOnDly_ET_7 { ExternalAccessible := 'False'; ExternalVisible := 'False'; ExternalWritable := 'False'} : Time;
      IEC_TimerOnDly_ET_8 { ExternalAccessible := 'False'; ExternalVisible := 'False'; ExternalWritable := 'False'} : Time;
      IEC_TimerOnDly_ET_9 { ExternalAccessible := 'False'; ExternalVisible := 'False'; ExternalWritable := 'False'} : Time;
      IEC_TimerOnDly_ET_10 { ExternalAccessible := 'False'; ExternalVisible := 'False'; ExternalWritable := 'False'} : Time;
      IEC_TimerOnDly_DN_1 { ExternalAccessible := 'False'; ExternalVisible := 'False'; ExternalWritable := 'False'} : Bool;
      IEC_TimerOnDly_DN_2 { ExternalAccessible := 'False'; ExternalVisible := 'False'; ExternalWritable := 'False'} : Bool;
      IEC_TimerOnDly_DN_3 { ExternalAccessible := 'False'; ExternalVisible := 'False'; ExternalWritable := 'False'} : Bool;
      IEC_TimerOnDly_DN_4 { ExternalAccessible := 'False'; ExternalVisible := 'False'; ExternalWritable := 'False'} : Bool;
      IEC_TimerOnDly_DN_5 { ExternalAccessible := 'False'; ExternalVisible := 'False'; ExternalWritable := 'False'} : Bool;
      IEC_TimerOnDly_DN_6 { ExternalAccessible := 'False'; ExternalVisible := 'False'; ExternalWritable := 'False'} : Bool;
      IEC_TimerOnDly_DN_7 { ExternalAccessible := 'False'; ExternalVisible := 'False'; ExternalWritable := 'False'} : Bool;
      IEC_TimerOnDly_DN_8 { ExternalAccessible := 'False'; ExternalVisible := 'False'; ExternalWritable := 'False'} : Bool;
      IEC_TimerOnDly_DN_9 { ExternalAccessible := 'False'; ExternalVisible := 'False'; ExternalWritable := 'False'} : Bool;
      IEC_TimerOnDly_DN_10 { ExternalAccessible := 'False'; ExternalVisible := 'False'; ExternalWritable := 'False'} : Bool;
      LeftLegIndex { ExternalAccessible := 'False'; ExternalVisible := 'False'; ExternalWritable := 'False'} : Int;
      RightLegIndex { ExternalAccessible := 'False'; ExternalVisible := 'False'; ExternalWritable := 'False'} : Int;
      LeftLegsArrayIndex { ExternalAccessible := 'False'; ExternalVisible := 'False'; ExternalWritable := 'False'} : Array[1..6] of Bool;
      RightLegsArrayIndex { ExternalAccessible := 'False'; ExternalVisible := 'False'; ExternalWritable := 'False'} : Array[1..6] of Bool;
      ButtomFasting_Activated { ExternalAccessible := 'False'; ExternalVisible := 'False'; ExternalWritable := 'False'} : Bool;
      Helix_Activated { ExternalAccessible := 'False'; ExternalVisible := 'False'; ExternalWritable := 'False'} : Bool;
   END_VAR
   VAR RETAIN
      DlyToFinishButtonFasten { S7_SetPoint := 'True'} : Int := 50;
   END_VAR
   VAR 
      MovingUPDOWN_Activated { ExternalAccessible := 'False'; ExternalVisible := 'False'; ExternalWritable := 'False'} : Bool;
      MoveUPDOWN_LevoSpredaj { ExternalAccessible := 'False'; ExternalVisible := 'False'; ExternalWritable := 'False'} : Bool;
      MoveUPDOWN_LevoZadaj { ExternalAccessible := 'False'; ExternalVisible := 'False'; ExternalWritable := 'False'} : Bool;
      MoveUPDOWN_DESNOSpredaj { ExternalAccessible := 'False'; ExternalVisible := 'False'; ExternalWritable := 'False'} : Bool;
      MoveUPDOWN_DESNOZadaj { ExternalAccessible := 'False'; ExternalVisible := 'False'; ExternalWritable := 'False'} : Bool;
   END_VAR
   VAR RETAIN
      DlyToRotateOpposite { S7_SetPoint := 'True'} : Int := 60;
      WaitTimeBeforeMoveDown { S7_SetPoint := 'True'} : Int := 100;
   END_VAR
   VAR 
      WaitLevoSpredaj { ExternalAccessible := 'False'; ExternalVisible := 'False'; ExternalWritable := 'False'} : Bool;
      WaitLevoZadaj { ExternalAccessible := 'False'; ExternalVisible := 'False'; ExternalWritable := 'False'} : Bool;
      WaitDesnoSpredaj { ExternalAccessible := 'False'; ExternalVisible := 'False'; ExternalWritable := 'False'} : Bool;
      WaitDesnoZadaj { ExternalAccessible := 'False'; ExternalVisible := 'False'; ExternalWritable := 'False'} : Bool;
      FOTOCELICA_LOC_TRAK_LEVO1_Latch { ExternalAccessible := 'False'; ExternalVisible := 'False'; ExternalWritable := 'False'} : Bool;
      FOTOCELICA_LOC_TRAK_LEVO2_Latch { ExternalAccessible := 'False'; ExternalVisible := 'False'; ExternalWritable := 'False'} : Bool;
      FOTOCELICA_LOC_TRAK_DESNO1_Latch { ExternalAccessible := 'False'; ExternalVisible := 'False'; ExternalWritable := 'False'} : Bool;
      FOTOCELICA_LOC_TRAK_DESNO2_Latch { ExternalAccessible := 'False'; ExternalVisible := 'False'; ExternalWritable := 'False'} : Bool;
   END_VAR
   VAR RETAIN
      WEndTimeToRemovePlate { S7_SetPoint := 'True'} : Int := 20;
   END_VAR
   VAR 
      LeftLegIndexOLD { ExternalAccessible := 'False'; ExternalVisible := 'False'; ExternalWritable := 'False'} : Int;
      RightLegIndexOLD { ExternalAccessible := 'False'; ExternalVisible := 'False'; ExternalWritable := 'False'} : Int;
      StartReleaseTimer1 { ExternalAccessible := 'False'; ExternalVisible := 'False'; ExternalWritable := 'False'} : Bool;
      StartReleaseTimer2 { ExternalAccessible := 'False'; ExternalVisible := 'False'; ExternalWritable := 'False'} : Bool;
      FOTOCELICA_LEVO_SPREDAJ_LATCH { ExternalAccessible := 'False'; ExternalVisible := 'False'; ExternalWritable := 'False'} : Bool;
      FOTOCELICA_LEVO_ZADAJ_LATCH { ExternalAccessible := 'False'; ExternalVisible := 'False'; ExternalWritable := 'False'} : Bool;
      FOTOCELICA_DESNO_SPREDAJ_LATCH { ExternalAccessible := 'False'; ExternalVisible := 'False'; ExternalWritable := 'False'} : Bool;
      FOTOCELICA_DESNO_ZADAJ_LATCH { ExternalAccessible := 'False'; ExternalVisible := 'False'; ExternalWritable := 'False'} : Bool;
   END_VAR
   VAR RETAIN
      DlyToStartButtomFasten { S7_SetPoint := 'True'} : Int := 50;
   END_VAR
   VAR 
      EndLevoSpredaj { ExternalAccessible := 'False'; ExternalVisible := 'False'; ExternalWritable := 'False'} : Bool;
      EndLevoZadaj { ExternalAccessible := 'False'; ExternalVisible := 'False'; ExternalWritable := 'False'} : Bool;
      EndDesnoSpredaj { ExternalAccessible := 'False'; ExternalVisible := 'False'; ExternalWritable := 'False'} : Bool;
      EndDesnoZadaj { ExternalAccessible := 'False'; ExternalVisible := 'False'; ExternalWritable := 'False'} : Bool;
   END_VAR
   VAR RETAIN
      DlyToInitRunTrakVijac { ExternalAccessible := 'False'; ExternalVisible := 'False'; ExternalWritable := 'False'; S7_SetPoint := 'True'} : Int := 50;
   END_VAR
   VAR 
      LegsReadyOnPosToHelix { ExternalAccessible := 'False'; ExternalVisible := 'False'; ExternalWritable := 'False'} : Bool;
      VpenjanjeDnaActived { ExternalAccessible := 'False'; ExternalVisible := 'False'; ExternalWritable := 'False'} : Bool;
   END_VAR
   VAR RETAIN
      RegimeHelix { S7_SetPoint := 'True'} : Bool;
      TotalButtomPlateCounter : UDInt;
   END_VAR
   VAR 
      DetectStartButtom { ExternalAccessible := 'False'; ExternalVisible := 'False'; ExternalWritable := 'False'} : Bool;
      InsertNewButtom { ExternalAccessible := 'False'; ExternalVisible := 'False'; ExternalWritable := 'False'} : USInt;
   END_VAR
   VAR RETAIN
      TimeoutToEndHelix { ExternalAccessible := 'False'; ExternalVisible := 'False'; ExternalWritable := 'False'; S7_SetPoint := 'True'} : UInt := 80;
   END_VAR
   VAR 
      FirstButtom { ExternalAccessible := 'False'; ExternalVisible := 'False'; ExternalWritable := 'False'} : Bool;
   END_VAR

   VAR_TEMP 
      i : Int;
      i1 : Int;
      i2 : Int;
      i3 : Int;
      i4 : Int;
      i5 : Int;
      i6 : Int;
      i7 : Int;
      i8 : Int;
      i9 : Int;
      i10 : Int;
   END_VAR

   VAR CONSTANT 
      ReleaseValOnBeltSepaTime : Int := 20;
      PLIIndex : Int := 1;
   END_VAR


BEGIN
	// Initialize variables
	#i1   := #PLIIndex;                          // 1
	#i2   := #PLIIndex + "MaxPLITimersIndex";    // 5
	#i3   := #PLIIndex + 2*"MaxPLITimersIndex";  // 9
	#i4   := #PLIIndex + 3*"MaxPLITimersIndex";  // 13
	#i5   := #PLIIndex + 4*"MaxPLITimersIndex";  // 17
	#i6   := #PLIIndex + 5*"MaxPLITimersIndex";  // 21
	#i7   := #PLIIndex + 6*"MaxPLITimersIndex";  // 25
	#i8   := #PLIIndex + 7*"MaxPLITimersIndex";  // 29
	#i9   := #PLIIndex + 8*"MaxPLITimersIndex";  // 33
	#i10  := #PLIIndex + 9*"MaxPLITimersIndex";  // 37
	
	// Check alarms
	#AlarmPresent := 0;
	FOR #i := 1 TO 32 DO
	  IF "dbAlarms".PLI[#PLIIndex, #i] THEN
	    #AlarmPresent := 1;
	    // #StartCmd     := False;
	  END_IF;
	  IF "AlarmAck" THEN
	    "dbAlarms".PLI[#PLIIndex, #i] := 0;
	  END_IF;
	END_FOR;
	
	// Timers section
	#IEC_TimerOnDly_DN_1 := 0;
	#IEC_TimerOnDly_1(IN := #CurrentStep = 1 AND NOT #InitPosition,
	                  R := #CurrentStep <> 1,
	                  PT := T#3s,
	                  Q => #IEC_TimerOnDly_DN_1,
	                  ET => #IEC_TimerOnDly_ET_1);
	
	// PHASE STATUS
	#PhaseStatus := 0;
	IF #CurrentStep >= 1 AND #StartCmd THEN
	  #PhaseStatus := 5;
	END_IF;
	IF #CurrentStep >= 1 AND NOT #StartCmd THEN
	  #PhaseStatus := 7;
	END_IF;
	IF #CurrentStep >= 1 AND #AlarmPresent THEN
	  #PhaseStatus := 6;
	END_IF;
	
	// Stop phase if START CMD=0
	IF NOT #StartCmd AND #CurrentStep > 0 THEN
	  #CurrentStep := 0;
	END_IF;
	
	CASE #CurrentStep OF
	  0: // Sequence permissives
	  "dbTimers".Num[#i1].EE    := False;
	
	  IF (#StartCmd AND TRUE) THEN // Local  mode
	    IF #PhaseStatus=0 THEN
	
	      // BEGIN - Init variable only at the begining
	      #LeftLegIndex  := 0;  // Reset at the begining only, next filling new legs when moved away from #Y12_VijaLocev_Lev
	      #LeftLegsArrayIndex[1] := False;
	      #LeftLegsArrayIndex[2] := False;
	      #LeftLegsArrayIndex[3] := False;
	      #LeftLegsArrayIndex[4] := False;
	      #LeftLegsArrayIndex[5] := False;
	      #LeftLegsArrayIndex[6] := False;
	  
	      #RightLegIndex := 0;  // Reset at the begining only, next filling new legs when moved away from #Y8_VijaLocev_Des 
	      #RightLegsArrayIndex[1] := False;
	      #RightLegsArrayIndex[2] := False;
	      #RightLegsArrayIndex[3] := False;
	      #RightLegsArrayIndex[4] := False;
	      #RightLegsArrayIndex[5] := False;
	      #RightLegsArrayIndex[6] := False;
	
	      #LegsReadyOnPosToHelix := False;
	
	      #InitPosition       := False;
	      #InsertNewButtom    := 0;
	
	      #FOTOCELICA_LOC_TRAK_LEVO1_Latch  := False;
	      #FOTOCELICA_LOC_TRAK_LEVO2_Latch  := False;
	      #FOTOCELICA_LOC_TRAK_DESNO1_Latch := False;
	      #FOTOCELICA_LOC_TRAK_DESNO2_Latch := False;
	      // END - Init variable only at the begining
	      
	      #FirstButtom := True;
	
	      #CurrentStep := 1;
	    END_IF;   
	  END_IF;
	
	  1: // Check initial positions
	    #InitPosition := (
	                       (#LeftLegIndex=0 AND #RightLegIndex=0)
	                       AND
	                       (
	                         ("dbDigitalSensors".MESTO_VIJAC_STOP_LEVO_ZAD_NAPREJ.InputF AND "dbDigitalSensors".MESTO_VIJAC_STOP_DESNO_ZAD_NAPREJ.InputF) AND
	                          // Begin with legs already present on positions for helixs FOTOCELICA_VIJACENJE_LEVO_ZADAJ,FOTOCELICA_VIJACENJE_LEVO_SPREDAJ
	                          // FOTOCELICA_VIJACENJE_DESNOZADAJ, FOTOCELICA_VIJACENJE_DESNOSPREDAJ
	                         (*
	                         (NOT "dbDigitalSensors".FOTOCELICA_VIJACENJE_LEVO_ZADAJ.InputF AND NOT "dbDigitalSensors".FOTOCELICA_VIJACENJE_LEVO_SPREDAJ.InputF AND 
	                         NOT "dbDigitalSensors".FOTOCELICA_VIJACENJE_DESNOZADAJ.InputF AND NOT "dbDigitalSensors".FOTOCELICA_VIJACENJE_DESNOSPREDAJ.InputF)
	                         AND
	                         *)
	                         ("dbDigitalSensors".MESTO_VIJACENJE_LEVO_ZAD_DVIG_DOL.InputF AND "dbDigitalSensors".MESTO_VIJACENJE_LEVO_SPRED_DVIG_DOL.InputF AND
	                         "dbDigitalSensors".MESTO_VIJACENJE_DESNO_ZAD_DVIG_DOL.InputF AND "dbDigitalSensors".MESTO_VIJACENJE_DESNO_SPRED_DVIG_DOL.InputF)
	                         AND
	                         ("dbDigitalSensors".MESTO_VIJACENJE_LEVO_ZAD_CENT_NARAZEN.InputF AND "dbDigitalSensors".MESTO_VIJACENJE_LEVO_SPRED_CENT_NARAZEN.InputF AND 
	                         "dbDigitalSensors".MESTO_VIJACENJE_DESNO_ZAD_CENT_NARAZEN.InputF AND "dbDigitalSensors".MESTO_VIJACENJE_DESNO_SPRED_CENT_NARAZEN.InputF)
	                         AND
	                         ("dbDigitalSensors".VPENJANJE_DNA_LEVO_ZADAJ_GOR.InputF AND "dbDigitalSensors".VPENJANJE_DNA_LEVO_SPREDAJ_GOR.InputF AND 
	                         "dbDigitalSensors".VPENJANJE_DNA_DESNO_ZADAJ_GOR.InputF AND "dbDigitalSensors".VPENJANJE_DNA_DESNO_SPREDAJ_GOR.InputF)
	                       )
	                     )
	                     OR 
	                     (
	                       (#LeftLegIndex=2 AND #RightLegIndex=2)
	                       AND
	                       (
	                         ("dbDigitalSensors".MESTO_VIJACENJE_LEVO_ZAD_DVIG_DOL.InputF AND "dbDigitalSensors".MESTO_VIJACENJE_LEVO_SPRED_DVIG_DOL.InputF AND
	                         "dbDigitalSensors".MESTO_VIJACENJE_DESNO_ZAD_DVIG_DOL.InputF AND "dbDigitalSensors".MESTO_VIJACENJE_DESNO_SPRED_DVIG_DOL.InputF)
	                         AND
	                         ("dbDigitalSensors".VPENJANJE_DNA_LEVO_ZADAJ_GOR.InputF AND "dbDigitalSensors".VPENJANJE_DNA_LEVO_SPREDAJ_GOR.InputF AND 
	                         "dbDigitalSensors".VPENJANJE_DNA_DESNO_ZADAJ_GOR.InputF AND "dbDigitalSensors".VPENJANJE_DNA_DESNO_SPREDAJ_GOR.InputF)
	                       )
	                     );
	
	    IF #InitPosition THEN
	      #CurrentStep := 2;
	    END_IF;
	
	  2: // Check, if helixs already present on positions: FOTOCELICA_LOC_TRAK_LEVO1 | FOTOCELICA_LOC_TRAK_LEVO2 | FOTOCELICA_LOC_TRAK_DESNO1 | FOTOCELICA_LOC_TRAK_DESNO2
	    // OR on positions: FOTOCELICA_VIJACENJE_LEVO_SPREDAJ | FOTOCELICA_VIJACENJE_LEVO_ZADAJ | FOTOCELICA_VIJACENJE_DESNO_SPREDAJ | FOTOCELICA_VIJACENJE_DESNO_ZADAJ
	    
	    // REGION CENTRIRANJE AT BEGIN v funkciji v primeru že narejena vijačenja in da ni bila nobena nogica privijačena v pladenj
	    // in je bila vrnjena pred fotocelice na pozicijah za start vijačenja
	    (*
	    REGION CENTRIRANJE AT BEGIN
	    // *************** BEGIN - Stop ZADAJ and centring *************** //
	    // Stop moving second leg, with open valve
	    IF #LeftLegIndex=1 OR #LeftLegIndex=2 THEN
	      #Y13_VijaStop_LevZad.AutoON := True;
	    END_IF;
	    IF #LeftLegsArrayIndex[1] THEN
	      #Y15_Centri_LevSpr.AutoON := TRUE;
	    END_IF;
	    IF #LeftLegsArrayIndex[2] THEN
	      #Y14_Centri_LevZad.AutoON := TRUE;
	    END_IF;
	
	    // Stop moving second leg, with open valve
	    IF #RightLegIndex=1 OR #RightLegIndex=2 THEN
	      #Y9_VijaStop_DesZad.AutoON := True;
	    END_IF;
	    IF #RightLegsArrayIndex[1] THEN
	      #Y11_Centri_DesSpr.AutoON := TRUE;
	    END_IF;
	    IF #RightLegsArrayIndex[2] THEN
	      #Y10_Centri_DesZad.AutoON := TRUE;
	    END_IF;
	    // **************** END - Stop ZADAJ and centring **************** //  
	    END_REGION CENTRIRANJE
	    *)
	
	    "dbTimers".Num[#i1].FR    := False;
	    "dbTimers".Num[#i2].FR    := False;
	    "dbTimers".Num[#i3].FR    := False;
	    "dbTimers".Num[#i4].FR    := False;
	    "dbTimers".Num[#i1].EE    := True;
	    "dbTimers".Num[#i1].PRE   := #DlyToInitRunTrakVijac;
	
	    #VKLOP_M_TRAKA_VIJACNIKA.AutoON := True; // See "ph_LegsShifter_2_DB".#StartCmd := True in op_ButtonHelix_3 (Run #VKLOP_M_TRAKA_VIJACNIKA, before checking if legs present in ph_LegsShifter_2, CurrentStep=3)
	
	    // Next step
	    IF ("dbTimers".Num[#i1].EE AND "dbTimers".Num[#i1].DN) THEN
	      // Check if all legs ready on positions to move motors UP and start with execute helix
	      IF #LeftLegIndex=2 OR #RightLegIndex=2 THEN
	        #LegsReadyOnPosToHelix := True;
	      END_IF;
	      IF #FirstButtom THEN
	        // 20210512_PRA Added to start with helixs already present
	        IF "dbDigitalSensors".FOTOCELICA_VIJACENJE_LEVO_ZADAJ.InputF AND "dbDigitalSensors".FOTOCELICA_VIJACENJE_LEVO_SPREDAJ.InputF THEN
	          #LeftLegIndex := 2;
	        END_IF;
	        IF "dbDigitalSensors".FOTOCELICA_VIJACENJE_DESNOZADAJ.InputF AND "dbDigitalSensors".FOTOCELICA_VIJACENJE_DESNOSPREDAJ.InputF THEN
	          #RightLegIndex := 2;
	        END_IF;
	      END_IF;
	      // 20210512_PRA
	      #CurrentStep := 3;
	    END_IF;
	
	  3: // Preveri stanje nogic na poziciji za vijačenje
	     // DOVOLJENO STANJE:
	     // 1. Prisotne vse 4. nogice na poziciji za vijačenje (po koncu neuspešnega vijačenja nogic. Nogice niso bile privijačene is čakajo na poziciji vijačenja - po koncu CurrentStep=10)
	     // 2. Manjkajo vse 4. nogice na poziciji za vijačenje (po STARTu iz začetnega koraka; CurrentStep=0)
	    #CurrentStep := 5;
	
	  5: // Init variables
	
	    // BEGIN - Init variable for each next buttom
	    "dbTimers".Num[#i1].EE    := False;
	    "dbTimers".Num[#i2].EE    := False;
	    "dbTimers".Num[#i3].EE    := False;
	    "dbTimers".Num[#i4].EE    := False;
	    "dbTimers".Num[#i5].EE    := False;
	    "dbTimers".Num[#i6].EE    := False;
	    "dbTimers".Num[#i7].EE    := False;
	    "dbTimers".Num[#i8].EE    := False;
	    "dbTimers".Num[#i9].EE    := False;
	    "dbTimers".Num[#i10].EE   := False; // Used for delay time. Delay time for button plate present on helix positions (see: #ButtonFasting_Activated)
	    
	    "dbTimers".Num[#i1].DN    := False;
	    "dbTimers".Num[#i2].DN    := False;
	    "dbTimers".Num[#i3].DN    := False;
	    "dbTimers".Num[#i4].DN    := False;
	    "dbTimers".Num[#i5].DN    := False;
	    "dbTimers".Num[#i6].DN    := False;
	    "dbTimers".Num[#i7].DN    := False;
	    "dbTimers".Num[#i8].DN    := False;
	    "dbTimers".Num[#i9].DN    := False;
	    "dbTimers".Num[#i10].DN   := False;
	
	    "dbTimers".Num[#i1].FR    := False;
	    "dbTimers".Num[#i2].FR    := False;
	    "dbTimers".Num[#i3].FR    := False;
	    "dbTimers".Num[#i4].FR    := False;
	    "dbTimers".Num[#i5].FR    := False;
	    "dbTimers".Num[#i6].FR    := False;
	    "dbTimers".Num[#i7].FR    := False;
	    "dbTimers".Num[#i8].FR    := False;
	    "dbTimers".Num[#i9].FR    := False;
	    "dbTimers".Num[#i10].FR   := False;
	
	    #ButtomFasting_Activated  := False;
	    #Helix_Activated          := False;
	    #MovingUPDOWN_Activated   := False;
	
	    #WaitLevoSpredaj          := False;
	    #MoveUPDOWN_LevoSpredaj   := False;
	    #WaitLevoZadaj            := False;
	    #MoveUPDOWN_LevoZadaj     := False;
	    #WaitDesnoSpredaj         := False;
	    #MoveUPDOWN_DESNOSpredaj  := False;
	    #WaitDesnoZadaj           := False;
	    #MoveUPDOWN_DESNOZadaj    := False;
	    #EndLevoSpredaj           := False;
	    #EndLevoZadaj             := False;
	    #EndDesnoSpredaj          := False;
	    #EndDesnoZadaj            := False;
	
	    #FOTOCELICA_LEVO_SPREDAJ_LATCH  := False;
	    #FOTOCELICA_LEVO_ZADAJ_LATCH    := False;
	    #FOTOCELICA_DESNO_SPREDAJ_LATCH := False;
	    #FOTOCELICA_DESNO_ZADAJ_LATCH   := False;
	    
	    #StartReleaseTimer1 := FALSE;
	    #StartReleaseTimer2 := FALSE;
	
	    // Check PRA_20210425 "ph_LegsShifter_2_DB".LeftLegIndex  := 0;
	    // Check PRA_20210425 "ph_LegsShifter_2_DB".RightLegIndex := 0;
	
	    "TestINT_01" := 0;
	    "IND_VIJAC_LEVO_NAPREJ"   := False;
	    "IND_VIJAC_LEVO_NAZAJ"    := False;
	    "IND_VIJAC_DES_NAPREJ"    := False;
	    "IND_VIJAC_DES_NAZAJ"     := False;
	    
	    #VpenjanjeDnaActived := False;
	    #DetectStartButtom := False;
	    // END - Init variable for each next buttom
	    
	    #FirstButtom := False; // Clear NOT set #LeftLegIndex=2, #RightLegIndex=2
	
	    #CurrentStep := 10;
	  
	  10: // Main step - moving legs through legs conveyor and helix legs to the button plate
	    // ******************* BEGIN - ALARM STATE *********** // 
	    IF NOT #AlarmPresent THEN
	      "dbTimers".Num[#i1].FR    := False;
	      "dbTimers".Num[#i2].FR    := False;
	      "dbTimers".Num[#i3].FR    := False;
	      "dbTimers".Num[#i4].FR    := False;
	      "dbTimers".Num[#i5].FR    := False;
	      "dbTimers".Num[#i6].FR    := False;
	      "dbTimers".Num[#i7].FR    := False;
	      "dbTimers".Num[#i8].FR    := False;
	      "dbTimers".Num[#i10].FR   := False;
	    ELSE
	      "dbTimers".Num[#i1].FR    := True;
	      "dbTimers".Num[#i2].FR    := True;
	      "dbTimers".Num[#i3].FR    := True;
	      "dbTimers".Num[#i4].FR    := True;
	      "dbTimers".Num[#i5].FR    := True;
	      "dbTimers".Num[#i6].FR    := True;
	      "dbTimers".Num[#i7].FR    := True;
	      "dbTimers".Num[#i8].FR    := True;
	      "dbTimers".Num[#i10].FR   := True;
	    END_IF;
	    // ********************* END - ALARM STATE ************ // 
	
	    IF NOT #AlarmPresent AND NOT #Helix_Activated THEN // Run #VKLOP_M_TRAKA_VIJACNIKA when helix is not active
	      #VKLOP_M_TRAKA_VIJACNIKA.AutoON := True; 
	    END_IF;
	
	    REGION RELEASE HELIXS ON VIJACNJI DEL
	    IF NOT #ButtomFasting_Activated THEN // Prevent to use timer[#1] at the same time (Legs moving on conveyor+Start moving UP/DOWN and with helix)
	      // *************** BEGIN - Legs moving on conveyor - left side *************** //
	      (*
	      IF (("dbDigitalSensors".START_LEVO_NA_VPENJANJU.OSR OR "dbDigitalSensors".START_DESNO_NA_VPENJANJU.OSR) AND
	          ("dbDigitalSensors".FOTOCELICA_LOC_TRAK_LEVO1.InputF AND "dbDigitalSensors".FOTOCELICA_LOC_TRAK_LEVO2.InputF // open first time when 2 legs infront and NO button plate present on helix positions
	           AND #LeftLegIndex = 0))
	           OR
	           ("dbDigitalSensors".FOTOCELICA_LOC_TRAK_LEVO1.InputF AND #LeftLegIndex=1 AND NOT #StartReleaseTimer1 AND "dbDigitalSensors".VIJACENJE_LEVO_1_NAPREJ.InputF)
	        THEN
	        #StartReleaseTimer1 := True;
	      END_IF;
	      *)
	      "StartCondToReleaseVijacenje1" := ("ph_LegsShifter_2_DB".LeftLegIndex=2 OR ("ph_LegsShifter_2_DB".LeftLegIndex=0 AND "dbDigitalSensors".FOTOCELICA_LOC_TRAK_LEVO1.InputF AND "dbDigitalSensors".FOTOCELICA_LOC_TRAK_LEVO2.InputF));
	      "StartCondToReleaseVijacenje2" := ("dbDigitalSensors".FOTOCELICA_LOC_TRAK_LEVO1.InputF AND "dbDigitalSensors".FOTOCELICA_LOC_TRAK_LEVO2.InputF AND #LeftLegIndex = 0);
	      "StartCondToReleaseVijacenje3" := ("dbDigitalSensors".FOTOCELICA_LOC_TRAK_LEVO1.InputF AND #LeftLegIndex=1 AND NOT #StartReleaseTimer1 AND "dbDigitalSensors".VIJACENJE_LEVO_1_NAPREJ.InputF);
	      (* // 20210512_PRA
	      IF  (("ph_LegsShifter_2_DB".LeftLegIndex=2 OR "ph_LegsShifter_2_DB".LeftLegIndex=0) AND // LeftLegIndex=2 -> naslednje spust s drce, LeftLegIndex=0 -> prvi spust s drce
	          ("dbDigitalSensors".MESTO_VIJACENJE_LEVO_SPRED_DVIG_DOL.InputF AND "dbDigitalSensors".MESTO_VIJACENJE_LEVO_ZAD_DVIG_DOL.InputF AND "dbMotors".VKLOP_M_TRAKA_VIJACNIKA.XS))
	          AND
	          (
	          // ("dbDigitalSensors".FOTOCELICA_LOC_TRAK_LEVO1.InputF AND "dbDigitalSensors".FOTOCELICA_LOC_TRAK_LEVO2.InputF AND #LeftLegIndex = 0)
	          ("ph_LegsShifter_2_DB".LeftLegIndex=2 AND NOT #StartReleaseTimer1 AND #LeftLegIndex = 0)
	          OR
	          // ("dbDigitalSensors".FOTOCELICA_LOC_TRAK_LEVO1.InputF AND #LeftLegIndex=1 AND NOT #StartReleaseTimer1 AND "dbDigitalSensors".VIJACENJE_LEVO_1_NAPREJ.InputF)
	          ("ph_LegsShifter_2_DB".LeftLegIndex=2 AND #LeftLegIndex=1 AND NOT #StartReleaseTimer1 AND "dbDigitalSensors".VIJACENJE_LEVO_1_NAPREJ.InputF)
	          )
	        THEN
	        #StartReleaseTimer1 := True;
	      END_IF;
	      *)
	      IF "dbDigitalSensors".FOTOCELICA_LOC_TRAK_LEVO1.InputF AND NOT #FOTOCELICA_LOC_TRAK_LEVO1_Latch THEN
	        #FOTOCELICA_LOC_TRAK_LEVO1_Latch := "dbDigitalSensors".FOTOCELICA_LOC_TRAK_LEVO1.InputF;
	      END_IF;
	      IF "dbDigitalSensors".FOTOCELICA_LOC_TRAK_LEVO2.InputF AND NOT #FOTOCELICA_LOC_TRAK_LEVO2_Latch AND #FOTOCELICA_LOC_TRAK_LEVO1_Latch THEN
	        #FOTOCELICA_LOC_TRAK_LEVO2_Latch := "dbDigitalSensors".FOTOCELICA_LOC_TRAK_LEVO2.InputF;
	      END_IF;
	
	      IF  (("ph_LegsShifter_2_DB".LeftLegIndex=2 AND #LeftLegIndex<>2) AND // For first buttom not need to prepare new helix if helixs already ready on helix positions 
	          ("dbDigitalSensors".MESTO_VIJACENJE_LEVO_SPRED_DVIG_DOL.InputF AND "dbDigitalSensors".MESTO_VIJACENJE_LEVO_ZAD_DVIG_DOL.InputF AND "dbMotors".VKLOP_M_TRAKA_VIJACNIKA.XS))
	          AND
	          (
	          (NOT #StartReleaseTimer1 AND #LeftLegIndex=0 AND #FOTOCELICA_LOC_TRAK_LEVO1_Latch)
	          OR
	          (NOT #StartReleaseTimer1 AND #LeftLegIndex=1 AND "dbDigitalSensors".VIJACENJE_LEVO_1_NAPREJ.InputF AND #FOTOCELICA_LOC_TRAK_LEVO2_Latch)
	          )
	        THEN
	        #StartReleaseTimer1 := True;
	      END_IF;
	
	      "dbTimers".Num[#i1].EE  := #StartReleaseTimer1;
	      "dbTimers".Num[#i1].PRE := #ReleaseValOnBeltSepaTime; // 1000 ms
	      IF "dbTimers".Num[#i1].EE AND "dbTimers".Num[#i1].DN THEN
	          "dbTimers".Num[#i1].EE := False;
	          "dbTimers".Num[#i1].DN := False;
	          #StartReleaseTimer1    := False;
	          #LeftLegIndex := #LeftLegIndex + 1; // Counts leg after it is moved away from FOTOCELICA_LOC_TRAK_LEVO1
	          IF #LeftLegIndex = 2 THEN
	            #FOTOCELICA_LOC_TRAK_LEVO1_Latch := False;
	            #FOTOCELICA_LOC_TRAK_LEVO2_Latch := False;
	            "ph_LegsShifter_2_DB".LeftLegIndex := 0; // Clear (#LeftLegIndex=0) if is #LeftLegIndex=2, inside phase ph_Helix_1
	          END_IF;
	      END_IF;
	      #Y12_VijaLocev_Lev.AutoON := ("dbTimers".Num[#i1].TT); // Release line until delay time expired
	      // *************** END - Legs moving on conveyor - left side *************** //  
	    
	      // *************** BEGIN - Legs moving on conveyor - right side *************** //
	      (*
	      IF (("dbDigitalSensors".START_LEVO_NA_VPENJANJU.OSR OR "dbDigitalSensors".START_DESNO_NA_VPENJANJU.OSR) AND
	          ("dbDigitalSensors".FOTOCELICA_LOC_TRAK_DESNO1.InputF AND "dbDigitalSensors".FOTOCELICA_LOC_TRAK_DESNO2.InputF // open first time when 2 legs infront and NO button plate present on helix positions
	           AND #RightLegIndex = 0))
	           OR
	           ("dbDigitalSensors".FOTOCELICA_LOC_TRAK_DESNO1.InputF AND #RightLegIndex=1 AND NOT #StartReleaseTimer2 AND "dbDigitalSensors".VIJACENJE_DESNO_1_NAPREJ.InputF)
	        THEN
	        #StartReleaseTimer2 := True;
	      END_IF;
	      *)
	      (* // 20210512_PRA
	      IF  (("ph_LegsShifter_2_DB".RightLegIndex=2 OR "ph_LegsShifter_2_DB".RightLegIndex=0) AND // RightLegIndex=2 -> naslednje spust s drce, RightLegIndex=0 -> prvi spust s drce
	          ("dbDigitalSensors".MESTO_VIJACENJE_DESNO_SPRED_DVIG_DOL.InputF AND "dbDigitalSensors".MESTO_VIJACENJE_DESNO_ZAD_DVIG_DOL.InputF AND "dbMotors".VKLOP_M_TRAKA_VIJACNIKA.XS))
	          AND
	          (
	          // ("dbDigitalSensors".FOTOCELICA_LOC_TRAK_DESNO1.InputF AND "dbDigitalSensors".FOTOCELICA_LOC_TRAK_DESNO2.InputF AND #RightLegIndex = 0)
	          ("ph_LegsShifter_2_DB".RightLegIndex=2 AND NOT #StartReleaseTimer2 AND #RightLegIndex = 0)
	          OR
	          ("ph_LegsShifter_2_DB".RightLegIndex=2 AND #RightLegIndex=1 AND NOT #StartReleaseTimer2 AND "dbDigitalSensors".VIJACENJE_DESNO_1_NAPREJ.InputF)
	          )
	        THEN
	        #StartReleaseTimer2 := True;
	      END_IF;
	      *)
	      IF "dbDigitalSensors".FOTOCELICA_LOC_TRAK_DESNO1.InputF AND NOT #FOTOCELICA_LOC_TRAK_DESNO1_Latch THEN
	        #FOTOCELICA_LOC_TRAK_DESNO1_Latch := "dbDigitalSensors".FOTOCELICA_LOC_TRAK_DESNO1.InputF;
	      END_IF;
	      IF "dbDigitalSensors".FOTOCELICA_LOC_TRAK_DESNO2.InputF AND NOT #FOTOCELICA_LOC_TRAK_DESNO2_Latch AND #FOTOCELICA_LOC_TRAK_DESNO1_Latch THEN
	        #FOTOCELICA_LOC_TRAK_DESNO2_Latch := "dbDigitalSensors".FOTOCELICA_LOC_TRAK_DESNO2.InputF;
	      END_IF;
	
	      IF  (("ph_LegsShifter_2_DB".RightLegIndex=2 AND #RightLegIndex<>2) AND // For first buttom not needed to prepare new helixs if helixs already ready on helix positions 
	          ("dbDigitalSensors".MESTO_VIJACENJE_DESNO_SPRED_DVIG_DOL.InputF AND "dbDigitalSensors".MESTO_VIJACENJE_DESNO_ZAD_DVIG_DOL.InputF AND "dbMotors".VKLOP_M_TRAKA_VIJACNIKA.XS))
	          AND
	          (
	          (NOT #StartReleaseTimer2 AND #RightLegIndex=0 AND #FOTOCELICA_LOC_TRAK_DESNO1_Latch)
	          OR
	          (NOT #StartReleaseTimer2 AND #RightLegIndex=1 AND "dbDigitalSensors".VIJACENJE_DESNO_1_NAPREJ.InputF AND #FOTOCELICA_LOC_TRAK_DESNO2_Latch)
	          )
	        THEN
	        #StartReleaseTimer2 := True;
	      END_IF;
	
	
	      "dbTimers".Num[#i2].EE  := #StartReleaseTimer2;
	      "dbTimers".Num[#i2].PRE := #ReleaseValOnBeltSepaTime; // 1000 ms
	      IF "dbTimers".Num[#i2].EE AND "dbTimers".Num[#i2].DN THEN
	          "dbTimers".Num[#i2].EE := False;
	          "dbTimers".Num[#i2].DN := False;
	          #StartReleaseTimer2    := False;
	          #RightLegIndex := #RightLegIndex + 1; // Counts leg after it is moved away from FOTOCELICA_LOC_TRAK_DESNO1
	          IF #RightLegIndex = 2 THEN
	            #FOTOCELICA_LOC_TRAK_DESNO1_Latch := False;
	            #FOTOCELICA_LOC_TRAK_DESNO2_Latch := False;
	            "ph_LegsShifter_2_DB".#RightLegIndex := 0; // Clear (#RightLegIndex=0) if is #RightLegIndex=2, inside phase ph_Helix_1
	          END_IF;
	      END_IF;
	
	      #Y8_VijaLocev_Des.AutoON := ("dbTimers".Num[#i2].TT); // Release line until delay time expired
	    END_IF; // #ButtonFasting_Activated - Prevent to use timer[#1] at the same time (Legs moving on conveyor+Start moving UP/DOWN and with helix)
	    // *************** END - Legs moving on conveyor - right side *************** //  
	    END_REGION RELEASE HELIXS ON VIJACNJI DEL
	
	    REGION CENTRIRANJE AT BEGIN
	    // *************** BEGIN - Stop ZADAJ and centring *************** //
	    // Do not centring, if previous buttom not been removed
	    IF (#InsertNewButtom=1) AND NOT "dbDigitalSensors".INDUKTIVEC_PRAVILNA_VLOZITEV_DNA_1.InputF AND
	      NOT "dbDigitalSensors".INDUKTIVEC_PRAVILNA_VLOZITEV_DNA_2.InputF THEN
	      "dbHMIUser".CurrMachineStep := 'Pritisni start vijacenja';
	      #InsertNewButtom := 2;
	    END_IF;
	    IF #RegimeHelix AND (#InsertNewButtom=2) AND "dbDigitalSensors".INDUKTIVEC_PRAVILNA_VLOZITEV_DNA_1.InputF AND
	      "dbDigitalSensors".INDUKTIVEC_PRAVILNA_VLOZITEV_DNA_2.InputF THEN
	      #InsertNewButtom := 3;
	    END_IF;
	
	    // Stop moving second leg, with open valve
	    // 20210506_PRA - Valve normal position changed. Without control signal "VijaStop_LevZad" is outside (helix stopped), With control signal "VijaStop_LevZad" is inside (helix not stopped)
	    // IF #LeftLegIndex=1 OR #LeftLegIndex=2 THEN
	    IF #LeftLegIndex=0 AND "dbTimers".Num[#i1].TT THEN
	      #Y13_VijaStop_LevZad.AutoON := True;
	    END_IF;
	    // Prepare front position for centring
	    IF "dbDigitalSensors".FOTOCELICA_VIJACENJE_LEVO_SPREDAJ.InputF AND NOT #FOTOCELICA_LEVO_SPREDAJ_LATCH THEN
	      #LeftLegsArrayIndex[1] := "dbDigitalSensors".FOTOCELICA_VIJACENJE_LEVO_SPREDAJ.InputF; // Reset, ko je vijacenje koncano
	      #FOTOCELICA_LEVO_SPREDAJ_LATCH := True;
	    END_IF;
	    IF #LeftLegsArrayIndex[1] AND #InsertNewButtom=0 AND #MoveUPDOWN_LevoSpredaj THEN
	      #Y15_Centri_LevSpr.AutoON := TRUE;
	    END_IF;
	    // Prepare rear position for centring
	    IF "dbDigitalSensors".FOTOCELICA_VIJACENJE_LEVO_ZADAJ.InputF AND NOT #FOTOCELICA_LEVO_ZADAJ_LATCH THEN
	      #LeftLegsArrayIndex[2] := "dbDigitalSensors".FOTOCELICA_VIJACENJE_LEVO_ZADAJ.InputF; // Reset, ko je vijacenje koncano
	      #FOTOCELICA_LEVO_ZADAJ_LATCH := True;
	    END_IF;
	    IF #LeftLegsArrayIndex[2] AND #InsertNewButtom=0 AND #MoveUPDOWN_LevoZadaj THEN
	      #Y14_Centri_LevZad.AutoON := TRUE;
	    END_IF;
	
